	#########################################################

		TransmissionType for TxPDOs and RxPDOs:

			0:										Event controlled and sychron (with SYNC-Object)
			1-240:									Cyclic and synchron (with SYNC-Object)
			254:									Producer specified
			255:									Acyclic and eventcontrolled 
			255 and EventTime = InhibitTime:	Cyclic

	#########################################################	*)


	(*************************************************** TxPDOs of CANOpenSlave ( MOVI-PLC ReceiveObjects) ***********************************************************)

	ExtConfig.NumberOfTxPDO				:= 4;		(*  TxPDO ---> CANopenSlave Transmit *)

	ExtConfig.TxPDO[1].EventTime			:= 100;		(* Slave: Index 0x18xx SubIndex 5: CycleTime in ms for CANopenSlave TXPDO *)
	ExtConfig.TxPDO[1].InhibitTime			:= 10;		(* Slave: Index 0x18xx SubIndex 3: InhibitTime in ms for CANopenSlave TxPDO *)
	ExtConfig.TxPDO[1].TransmissionType	:= 255;		(* Slave: Index 0x18xx SubIndex 2: TransmissionType for this TxPDO *)

	ExtConfig.TxPDO[2].EventTime			:= 100;		(* Slave: Index 0x18xx SubIndex 5: CycleTime in ms for CANopenSlave TXPDO *)
	ExtConfig.TxPDO[2].InhibitTime			:= 10;		(* Slave: Index 0x18xx SubIndex 3: InhibitTime in ms for CANopenSlave TxPDO *)
	ExtConfig.TxPDO[2].TransmissionType	:= 255;		(* Slave: Index 0x18xx SubIndex 2: TransmissionType for this TxPDO *)

	ExtConfig.TxPDO[3].EventTime			:= 100;		(* Slave: Index 0x18xx SubIndex 5: CycleTime in ms for CANopenSlave TXPDO *)
	ExtConfig.TxPDO[3].InhibitTime			:= 10;		(* Slave: Index 0x18xx SubIndex 3: InhibitTime in ms for CANopenSlave TxPDO *)
	ExtConfig.TxPDO[3].TransmissionType	:= 255;		(* Slave: Index 0x18xx SubIndex 2: TransmissionType for this TxPDO *)

	ExtConfig.TxPDO[4].EventTime			:= 100;		(* Slave: Index 0x18xx SubIndex 5: CycleTime in ms for CANopenSlave TXPDO *)
	ExtConfig.TxPDO[4].InhibitTime			:= 10;		(* Slave: Index 0x18xx SubIndex 3: InhibitTime in ms for CANopenSlave TxPDO *)
	ExtConfig.TxPDO[4].TransmissionType	:= 255;		(* Slave: Index 0x18xx SubIndex 2: TransmissionType for this TxPDO *)


	(*************************************************** RxPDOs of CANOpenSlave ( MOVI-PLC TransmitObjects) **********************************************************)

	ExtConfig.NumberOfRxPDO				:= 4;		(*  RxPDO ---> CANopenSlave Receive *)

	ExtConfig.RxPDO[1].EventTime			:= 100;		(* Master: CycleTime in ms for TransmitObjects (MOVI-PLC) *)
	ExtConfig.RxPDO[1].InhibitTime			:= 10;		(* Master: InhibitTime in ms for TransmitObjects (MOVI-PLC) *)
	ExtConfig.RxPDO[1].Length				:= 8;		(* Master: Length of this TransmitObject in bytes *)
	ExtConfig.RxPDO[1].TransmissionType	:= 255;		(* Slave: Index 0x14xx SubIndex 2: TransmissionType for this RxPDO *)

	ExtConfig.RxPDO[2].EventTime			:= 100;		(* Master: CycleTime in ms for TransmitObjects (MOVI-PLC) *)
	ExtConfig.RxPDO[2].InhibitTime			:= 10;		(* Master: InhibitTime in ms for TransmitObjects (MOVI-PLC) *)
	ExtConfig.RxPDO[2].Length				:= 8;		(* Master: Length of this TransmitObject in bytes *)
	ExtConfig.RxPDO[2].TransmissionType	:= 255;		(* Slave: Index 0x14xx SubIndex 2: TransmissionType for this RxPDO *)

	ExtConfig.RxPDO[3].EventTime			:= 100;		(* Master: CycleTime in ms for TransmitObjects (MOVI-PLC) *)
	ExtConfig.RxPDO[3].InhibitTime			:= 10;		(* Master: InhibitTime in ms for TransmitObjects (MOVI-PLC) *)
	ExtConfig.RxPDO[3].Length				:= 8;		(* Master: Length of this TransmitObject in bytes *)
	ExtConfig.RxPDO[3].TransmissionType	:= 255;		(* Slave: Index 0x14xx SubIndex 2: TransmissionType for this RxPDO *)

	ExtConfig.RxPDO[4].EventTime			:= 100;		(* Master: CycleTime in ms for TransmitObjects (MOVI-PLC) *)
	ExtConfig.RxPDO[4].InhibitTime			:= 10;		(* Master: InhibitTime in ms for TransmitObjects (MOVI-PLC) *)
	ExtConfig.RxPDO[4].Length				:= 8;		(* Master: Length of this TransmitObject in bytes *)
	ExtConfig.RxPDO[4].TransmissionType	:= 255;		(* Slave: Index 0x14xx SubIndex 2: TransmissionType for this RxPDO *)


	(***************************************************** Additional parameters to set in the CANOpenSlave  ***************************************************************)
(* Parameter for Cube67 DIO16 (56601) Submodul *)
	ExtConfig.stInitialParameter_COSlave.aIndex[1]			:= 16#2002;(*2. Module*)
	ExtConfig.stInitialParameter_COSlave.aSubIndex[1]	:= 2;(* Input function *)
	ExtConfig.stInitialParameter_COSlave.aBytes[1]		:= 1;
	ExtConfig.stInitialParameter_COSlave.aData[1]			:= 2#00000000;(* 0=Input, 1=Diag Input *)

	ExtConfig.stInitialParameter_COSlave.aIndex[2]			:= 16#2002;(*2. Module*)
	ExtConfig.stInitialParameter_COSlave.aSubIndex[2]	:= 3;(* Inpu/Output selection, channel 0..7,  Pin4*)
	ExtConfig.stInitialParameter_COSlave.aBytes[2]		:= 1;
	ExtConfig.stInitialParameter_COSlave.aData[2]			:= 2#00000000;(* 0=Input, 1=Output *)

	ExtConfig.stInitialParameter_COSlave.aIndex[3]			:= 16#2002;(*2. Module*)
	ExtConfig.stInitialParameter_COSlave.aSubIndex[3]	:= 4;(* Inpu/Output selection, channel 10..17,  Pin2*)
	ExtConfig.stInitialParameter_COSlave.aBytes[3]		:= 1;
	ExtConfig.stInitialParameter_COSlave.aData[3]			:= 2#00000000;(* 0=Input, 1=Output *)

	ExtConfig.stInitialParameter_COSlave.aIndex[4]			:= 16#2002;(*2. Module*)
	ExtConfig.stInitialParameter_COSlave.aSubIndex[4]	:= 5;(*Failsafe Mode, channel 0..7,  Pin4*)
	ExtConfig.stInitialParameter_COSlave.aBytes[4]		:= 1;
	ExtConfig.stInitialParameter_COSlave.aData[4]			:= 2#00000000;(* 0=last state, 1=Failsafe value *)

	ExtConfig.stInitialParameter_COSlave.aIndex[5]			:= 16#2002;(*2. Module*)
	ExtConfig.stInitialParameter_COSlave.aSubIndex[5]	:= 6;(*Failsafe Mode, channel 10..17,  Pin2*)
	ExtConfig.stInitialParameter_COSlave.aBytes[5]		:= 1;
	ExtConfig.stInitialParameter_COSlave.aData[5]			:= 2#00000000;(* 0=last state, 1=Failsafe value *)

	ExtConfig.stInitialParameter_COSlave.aIndex[6]			:= 16#2002;(*2. Module*)
	ExtConfig.stInitialParameter_COSlave.aSubIndex[6]	:= 7;(*Failsafe Value, channel 0..7,  Pin4*)
	ExtConfig.stInitialParameter_COSlave.aBytes[6]		:= 1;
	ExtConfig.stInitialParameter_COSlave.aData[6]			:= 2#00000000;(* 0=output low, 1=output high *)

	ExtConfig.stInitialParameter_COSlave.aIndex[7]			:= 16#2002;(*2. Module*)
	ExtConfig.stInitialParameter_COSlave.aSubIndex[7]	:= 8;(*Failsafe Value, channel 10..17,  Pin2*)
	ExtConfig.stInitialParameter_COSlave.aBytes[7]		:= 1;
	ExtConfig.stInitialParameter_COSlave.aData[7]			:= 2#00000000;(* 0=output low, 1=output high *)

	ExtConfig.stInitialParameter_COSlave.aIndex[8]			:= 16#2002;(*2. Module*)
	ExtConfig.stInitialParameter_COSlave.aSubIndex[8]	:= 9;(*function, channel 0..7,  Pin4*)
	ExtConfig.stInitialParameter_COSlave.aBytes[8]		:= 1;
	ExtConfig.stInitialParameter_COSlave.aData[8]			:= 2#00000000;(* 0=input no, 1=input nc *)

	ExtConfig.stInitialParameter_COSlave.aIndex[9]			:= 16#2002;(*2. Module*)
	ExtConfig.stInitialParameter_COSlave.aSubIndex[9]	:= 10;(*function, channel 10..17,  Pin2*)
	ExtConfig.stInitialParameter_COSlave.aBytes[9]		:= 1;
	ExtConfig.stInitialParameter_COSlave.aData[9]			:= 2#00000000;(* 0=input no, 1=input nc *)

(* Parameter for Cube67 DIO8 (56610) Submodul *)
	ExtConfig.stInitialParameter_COSlave.aIndex[10]		:= 16#2003;(*3 Module*)
	ExtConfig.stInitialParameter_COSlave.aSubIndex[10]	:= 2;(* Input function *)
	ExtConfig.stInitialParameter_COSlave.aBytes[10]		:= 1;
	ExtConfig.stInitialParameter_COSlave.aData[10]		:= 2#0000;(* 0=Input, 1=Diag Input *)

	ExtConfig.stInitialParameter_COSlave.aIndex[11]		:= 16#2003;(*3 Module*)
	ExtConfig.stInitialParameter_COSlave.aSubIndex[11]	:= 3;(* Inpu/Output selection, channel 0..3  Pin4*)
	ExtConfig.stInitialParameter_COSlave.aBytes[11]		:= 1;
	ExtConfig.stInitialParameter_COSlave.aData[11]		:= 2#0000;(* 0=Input, 1=Output *)

	ExtConfig.stInitialParameter_COSlave.aIndex[12]		:= 16#2003;(*3. Module*)
	ExtConfig.stInitialParameter_COSlave.aSubIndex[12]	:= 4;(* Inpu/Output selection, channel 10..13  Pin2*)
	ExtConfig.stInitialParameter_COSlave.aBytes[12]		:= 1;
	ExtConfig.stInitialParameter_COSlave.aData[12]		:= 2#0000;(* 0=Input, 1=Output *)

	ExtConfig.stInitialParameter_COSlave.aIndex[13]		:= 16#2003;(*3. Module*)
	ExtConfig.stInitialParameter_COSlave.aSubIndex[13]	:= 5;(*Failsafe Mode, channel 0..3,  Pin4*)
	ExtConfig.stInitialParameter_COSlave.aBytes[13]		:= 1;
	ExtConfig.stInitialParameter_COSlave.aData[13]		:= 2#0000;(* 0=last state, 1=Failsafe value *)

	ExtConfig.stInitialParameter_COSlave.aIndex[14]		:= 16#2003;(*3. Module*)
	ExtConfig.stInitialParameter_COSlave.aSubIndex[14]	:= 6;(*Failsafe Mode, channel 10..13,  Pin2*)
	ExtConfig.stInitialParameter_COSlave.aBytes[14]		:= 1;
	ExtConfig.stInitialParameter_COSlave.aData[14]		:= 2#0000;(* 0=last state, 1=Failsafe value *)

	ExtConfig.stInitialParameter_COSlave.aIndex[15]		:= 16#2003;(*3. Module*)
	ExtConfig.stInitialParameter_COSlave.aSubIndex[15]	:= 7;(*Failsafe Value, channel 0..3,  Pin4*)
	ExtConfig.stInitialParameter_COSlave.aBytes[15]		:= 1;
	ExtConfig.stInitialParameter_COSlave.aData[15]		:= 2#0000;(* 0=output low, 1=output high *)

	ExtConfig.stInitialParameter_COSlave.aIndex[16]		:= 16#2003;(*3. Module*)
	ExtConfig.stInitialParameter_COSlave.aSubIndex[16]	:= 8;(*Failsafe Value, channel 10..13,  Pin2*)
	ExtConfig.stInitialParameter_COSlave.aBytes[16]		:= 1;
	ExtConfig.stInitialParameter_COSlave.aData[16]		:= 2#0000;(* 0=output low, 1=output high *)

	ExtConfig.stInitialParameter_COSlave.aIndex[17]		:= 16#2003;(*3. Module*)
	ExtConfig.stInitialParameter_COSlave.aSubIndex[17]	:= 9;(*function, channel 0..3,  Pin4*)
	ExtConfig.stInitialParameter_COSlave.aBytes[17]		:= 1;
	ExtConfig.stInitialParameter_COSlave.aData[17]		:= 2#0000;(* 0=input no, 1=input nc *)

	ExtConfig.stInitialParameter_COSlave.aIndex[18]		:= 16#2003;(*3. Module*)
	ExtConfig.stInitialParameter_COSlave.aSubIndex[18]	:= 10;(*function, channel 10..13,  Pin2*)
	ExtConfig.stInitialParameter_COSlave.aBytes[18]		:= 1;
	ExtConfig.stInitialParameter_COSlave.aData[18]		:= 2#0000;(* 0=input no, 1=input nc *)

(* Parameter for Cube67 DIO8/DI8 (56691) Submodul *)
	ExtConfig.stInitialParameter_COSlave.aIndex[19]		:= 16#2001;(*1. Module*)
	ExtConfig.stInitialParameter_COSlave.aSubIndex[19]	:= 1;(* Inpu/Output selection, channel 0..7*)
	ExtConfig.stInitialParameter_COSlave.aBytes[19]		:= 1;
	ExtConfig.stInitialParameter_COSlave.aData[19]		:= 2#00000010;(* 0=Input, 1=Output *)

	ExtConfig.stInitialParameter_COSlave.aIndex[20]		:= 16#2001;(*1.. Module*)
	ExtConfig.stInitialParameter_COSlave.aSubIndex[20]	:= 2;(*Failsafe Mode, channel 0..7*)
	ExtConfig.stInitialParameter_COSlave.aBytes[20]		:= 1;
	ExtConfig.stInitialParameter_COSlave.aData[20]		:= 2#0000;(* 0=last state, 1=Failsafe value *)

	ExtConfig.stInitialParameter_COSlave.aIndex[21]		:= 16#2001;(*1. Module*)
	ExtConfig.stInitialParameter_COSlave.aSubIndex[21]	:= 3;(*Failsafe Value, channel 0..7*)
	ExtConfig.stInitialParameter_COSlave.aBytes[21]		:= 1;
	ExtConfig.stInitialParameter_COSlave.aData[21]		:= 2#0000;(* 0=output low, 1=output high *)

	ExtConfig.stInitialParameter_COSlave.aIndex[22]		:= 16#2001;(*1. Module*)
	ExtConfig.stInitialParameter_COSlave.aSubIndex[22]	:= 4;(*function, channel 0..7*)
	ExtConfig.stInitialParameter_COSlave.aBytes[22]		:= 1;
	ExtConfig.stInitialParameter_COSlave.aData[22]		:= 2#0000;(* 0=input no, 1=input nc *)

	ExtConfig.stInitialParameter_COSlave.aIndex[23]		:= 16#2001;(*1. Module*)
	ExtConfig.stInitialParameter_COSlave.aSubIndex[23]	:= 5;(*function, channel 10..17*)
	ExtConfig.stInitialParameter_COSlave.aBytes[23]		:= 1;
	ExtConfig.stInitialParameter_COSlave.aData[23]		:= 2#0000;(* 0=input no, 1=input nc *)


(*	(* Enable transmission of analog inputs *)
	ExtConfig.stInitialParameter_COSlave.aIndex[24]		:= 16#6423;
	ExtConfig.stInitialParameter_COSlave.aSubIndex[24]	:= 0;
	ExtConfig.stInitialParameter_COSlave.aBytes[24]		:= 1;
	ExtConfig.stInitialParameter_COSlave.aData[24]		:= 1;
*)

(* Enable automatic PDO mapping *)
	ExtConfig.stInitialParameter_COSlave.aIndex[24]		:= 16#2100;
	ExtConfig.stInitialParameter_COSlave.aSubIndex[24]	:= 0;
	ExtConfig.stInitialParameter_COSlave.aBytes[24]		:= 1;
	ExtConfig.stInitialParameter_COSlave.aData[24]		:= 1;

	(********************************************** Additional configuration. Default values are in most cases sufficient *****************************************************)

	ExtConfig.bIOHold						:= FALSE;
	ExtConfig.bNoSettingsDownload			:= FALSE;
	ExtConfig.bWaitBeforeOperational		:= FALSE;
	ExtConfig.bResetUnconditional			:= FALSE;

	ExtConfig.TimeOutHeartBeat				:= 250;				(* [ms] *)
(*	ExtConfig.DivTimeOutHeartBeat			:= 2;				(* Heartbeat Consumer = ExtConfig.TimeOutHeartBeat	 / ExtConfig.DivTimeOutHeartBeat *)*)
	ExtConfig.TimeOutNodeGuarding		:= 0;				(* [ms]. CAUTION ! DHP11B (MOVI-PLC basic) does NOT support NodeGuarding *)
	ExtConfig.TimeOutInitSequence			:= 10;				(* [seconds]. If the Init-Sequence takes longer than this TimeOut time --> Error *)
	ExtConfig.SyncCOBID						:= 0;				(* SyncObject ID for TransmissionType 0-240 (RxPDO). Usually 128. If 0, the ID will not be written *)
	ExtConfig.SyncTime						:= 0;				(* CycleTime for the SYNC-Object *)

	ExtConfig.TxPDO[1].COBID				:= 16#180;			(* In order to disable the use of RTR frames for the PDOs, set bit 30 = "RTR not allowed" *)
	ExtConfig.TxPDO[2].COBID				:= 16#280;			(* Ex. 16#4000_0280 *)
	ExtConfig.TxPDO[3].COBID				:= 16#380;
	ExtConfig.TxPDO[4].COBID				:= 16#480;			(* NOTE! These values are base values. The input "Address" will automatically be added *)
	ExtConfig.TxPDO[5].COBID				:= 16#680;
	ExtConfig.TxPDO[6].COBID				:= 16#1C0;
	ExtConfig.TxPDO[7].COBID				:= 16#2C0;
	ExtConfig.TxPDO[8].COBID				:= 16#3C0;
	ExtConfig.TxPDO[9].COBID				:= 16#4C0;
	ExtConfig.TxPDO[10].COBID				:= 16#6C0;

	ExtConfig.RxPDO[1].COBID				:= 16#200;
	ExtConfig.RxPDO[2].COBID				:= 16#300;
	ExtConfig.RxPDO[3].COBID				:= 16#400;
	ExtConfig.RxPDO[4].COBID				:= 16#500;
	ExtConfig.RxPDO[5].COBID				:= 16#780;
	ExtConfig.RxPDO[6].COBID				:= 16#240;
	ExtConfig.RxPDO[7].COBID				:= 16#340;
	ExtConfig.RxPDO[8].COBID				:= 16#440;
	ExtConfig.RxPDO[9].COBID				:= 16#540;
	ExtConfig.RxPDO[10].COBID				:= 16#7C0;

	Done := TRUE;

END_IF
END_FUNCTION_BLOCK

(* POU CodeSamples/CANopen/UniversalMaster/FB_Configuration_CANopenSlave_Phoenix_FLS_CO_DI8, ST *)
FUNCTION_BLOCK FB_Configuration_CANopenSlave_Phoenix_FLS_CO_DI8
VAR_INPUT
	Enable: BOOL; 			(* Activate config *)
END_VAR
VAR_OUTPUT
	Done: BOOL;				(* Config done *)
END_VAR
VAR_IN_OUT
	ExtConfig : MC_EXTENDEDCONFIG_COSLAVE	;
	(*
		########################################################################################################
			MC_EXTENDEDCONFIG_COSLAVE
		#########################################################################################################

						
		Variable								Value			Description
		-------------------------------------------------------------------------------------------------------------------------------------------------------------
		bWaitBeforeOperational 				BOOL;			When TRUE, after the coupler has been parameterized, it won't be switched in operational
																before this variable is FALSE. This can be used for example, to store the configuration with the FB
																MPLC_Universal_CANopen, with Service "SEWIOS_STORE", after a reset of the coppler 
		-------------------------------------------------------------------------------------------------------------------------------------------------------------
		bNoSettingsDownload 				BOOL;			TRUE : No configuration of the module. The configuration has to be done manually.
		-------------------------------------------------------------------------------------------------------------------------------------------------------------
		bResetUnconditional 					BOOL;			Even if the Connect FB isn't in fault it is possible to reset the bus coppler
		-------------------------------------------------------------------------------------------------------------------------------------------------------------
		bIOHold 								BOOL;			TRUE : Input data remain unchanged and the output data are not resetet also if the FB is in fault 
		-------------------------------------------------------------------------------------------------------------------------------------------------------------
		TimeOutHeartBeat					UINT;			If this value (ms) is different to zero, HeartbeatMode will be activated
		-------------------------------------------------------------------------------------------------------------------------------------------------------------
		TimeOutNodeGuarding 				UINT;			If this value (ms) is different to zero, NodeGuarding will be activated. 
																Caution ! The MOVI-PLC basic doesn´t support NodeGuarding 
		-------------------------------------------------------------------------------------------------------------------------------------------------------------
		TimeOutInitSequence					UINT;			Timeout for initialisation sequence (seconds) 
		-------------------------------------------------------------------------------------------------------------------------------------------------------------
		NumberOfRxPDO 					UINT;			Receive PDO : MOVI-PLC --> Slave  max. 32 
		-------------------------------------------------------------------------------------------------------------------------------------------------------------
		NumberOfTxPDO 						UINT;			Send PDO :      Slave --> MOVI-PLC  max 32 
		-------------------------------------------------------------------------------------------------------------------------------------------------------------	
		SyncTime 								USINT;			Cycle time of the sync telegram in ms. 
																Default = 0 : no sync will be started.
																If  SyncTime > 0, this FB initializes a sync telegram with the ID set at SyncCOBID. 
																The slave has to support synchronous communication 
		-------------------------------------------------------------------------------------------------------------------------------------------------------------
		SyncCOBID							UINT;			Index 1005h. ID of the sync telegram. Usually 16#80. IF 0, the ID won't be written.
		-------------------------------------------------------------------------------------------------------------------------------------------------------------
		SyncTimeOut 							INT := -1;		Index 1006h. Normally equal to SyncTime. 
																The slave usually set SyncTimeOut equal to SyncTime * 1.5. 
																If < 0, the index won't be written. 0 means no control over the sync interval 
		-------------------------------------------------------------------------------------------------------------------------------------------------------------
		stInitialParameter_COSlave 			MC_INITIALPARAMETER_COSLAVE;
												(*#################################################################
												With this struct, user defined parameters will be written to the BusCoupler after the
												initialization of the MPLC_ConnectUniversalSlave_CANopen. 
												Add the following code to your program to initialise the struct : 
												Example:
												Index 16#6423:	Activates the event-driven transmission of PDOs with analog inputs
												Index 16#3500:	Index from the manufacturer specific profile area
	
													stInitialParameter_COSlave.aIndex[1] := 16#6423;  	(* Index to write to *)
													stInitialParameter_COSlave.aSubIndex[1] := 0;   	(* SubIndex to write to *)
													stInitialParameter_COSlave.aBytes[1] := 1;   		(* Number of bytes to write  *)
													stInitialParameter_COSlave.aData[1] := 1;   			(* Data *)
	
													stInitialParameter_COSlave.aIndex[2] := 16#3500;  	(* Index to write to *)
													stInitialParameter_COSlave.aSubIndex[2] := 0;   	(* SubIndex to write to *)
													stInitialParameter_COSlave.aBytes[2] := 2;   		(* Number of bytes to write *)
													stInitialParameter_COSlave.aData[2] := 5;   			(* Data *)
	
												If there are more than 10 (DHP11B) or 64 (DHx41B) parameters to write, declare 
												NUMOF_INITIALPARAMETER in your program.
	
													VAR_GLOBAL CONSTANT
														NUMOF_INITIALPARAMETER : UDINT := 20;	
													END_VAR
	
												##################################################################*)
			-------------------------------------------------------------------------------------------------------------------------------------------------------------
		(* IDs of the PDO telegrams. The IDs are always calculated with the following IDs as a basis + the address of the bus coupler *)

		RxPDO 								ARRAY[1..32] OF MC_PDO_COSLAVE;			(* MOVI-PLC --> Slave *)
												(* := 16#200,16#300,16#400,16#500,16#780,16#240,16#340,16#440,16#540,16#7C0;	*)
		-------------------------------------------------------------------------------------------------------------------------------------------------------------
		TxPDO 								ARRAY[1..32] OF MC_PDO_COSLAVE; 			(* Slave --> MOVI-PLC *)
												(*:= 16#180,16#280,16#380,16#480,16#680,16#1C0,16#2C0,16#3C0,16#4C0,16#6C0;*)
	*)
END_VAR
IF Enable AND NOT Done THEN

	(*########################################################

		Configuration of CANopenSlave (Phoenix FLS CO DI8)
		
	#########################################################

		TransmissionType for TxPDOs and RxPDOs:

			0:										Event controlled and sychron (with SYNC-Object)
			1-240:									Cyclic and synchron (with SYNC-Object)
			254:									Producer specified
			255:									Acyclic and eventcontrolled 
			255 and EventTime = InhibitTime:	Cyclic

	#########################################################	*)


	(*************************************************** TxPDOs of CANOpenSlave ( MOVI-PLC ReceiveObjects) ***********************************************************)

	ExtConfig.NumberOfTxPDO				:= 1;		(*  TxPDO ---> CANopenSlave Transmit *)

	ExtConfig.TxPDO[1].EventTime			:= 0;		(* Slave: Index 0x18xx SubIndex 5: CycleTime in ms for CANopenSlave TXPDO *)
	ExtConfig.TxPDO[1].InhibitTime			:= 0;		(* Slave: Index 0x18xx SubIndex 3: InhibitTime in ms for CANopenSlave TxPDO *)
	ExtConfig.TxPDO[1].TransmissionType	:= 255;		(* Slave: Index 0x18xx SubIndex 2: TransmissionType for this TxPDO *)


	(*************************************************** RxPDOs of CANOpenSlave ( MOVI-PLC TransmitObjects) **********************************************************)

	ExtConfig.NumberOfRxPDO				:= 0;		(*  RxPDO ---> CANopenSlave Receive *)

(*	ExtConfig.RxPDO[1].EventTime			:= 0;		(* Master: CycleTime in ms for TransmitObjects (MOVI-PLC) *)
	ExtConfig.RxPDO[1].InhibitTime			:= 0;		(* Master: InhibitTime in ms for TransmitObjects (MOVI-PLC) *)
	ExtConfig.RxPDO[1].Length				:= 1;		(* Master: Length of this TransmitObject in bytes *)
	ExtConfig.RxPDO[1].TransmissionType	:= 255;		(* Slave: Index 0x14xx SubIndex 2: TransmissionType for this RxPDO *)
*)

	(***************************************************** Additional parameters to set in the CANOpenSlave  ***************************************************************)

(*	Example to write user defined parameters (i.e. Index 16#6200):
	
	ExtConfig.stInitialParameter_COSlave.aIndex[1]			:= 16#6200;
	ExtConfig.stInitialParameter_COSlave.aSubIndex[1]	:= 0;
	ExtConfig.stInitialParameter_COSlave.aBytes[1]		:= 1;
	ExtConfig.stInitialParameter_COSlave.aData[1]			:= 16#64;
*)

	(********************************************** Additional configuration. Default values are in most cases sufficient *****************************************************)

	ExtConfig.bIOHold						:= FALSE;
	ExtConfig.bNoSettingsDownload			:= FALSE;
	ExtConfig.bWaitBeforeOperational		:= FALSE;
	ExtConfig.bResetUnconditional			:= FALSE;

	ExtConfig.TimeOutHeartBeat				:= 0;				(* [ms] *)
	ExtConfig.TimeOutNodeGuarding		:= 400;				(* [ms]. CAUTION ! DHP11B (MOVI-PLC basic) does NOT support NodeGuarding *)
	ExtConfig.TimeOutInitSequence			:= 6;				(* [seconds]. If the Init-Sequence takes longer than this TimeOut time --> Error *)
	ExtConfig.SyncCOBID						:= 0;				(* SyncObject ID for TransmissionType 0-240 (RxPDO). Usually 128. If 0, the ID will not be written *)
	ExtConfig.SyncTime						:= 0;				(* CycleTime for the SYNC-Object *)

	ExtConfig.TxPDO[1].COBID				:= 16#180;			(* In order to disable the use of RTR frames for the PDOs, set bit 30 = "RTR not allowed" *)
	ExtConfig.TxPDO[2].COBID				:= 16#280;			(* Ex. 16#4000_0280 *)
	ExtConfig.TxPDO[3].COBID				:= 16#380;
	ExtConfig.TxPDO[4].COBID				:= 16#480;			(* NOTE! These values are base values. The input "Address" will automatically be added *)
	ExtConfig.TxPDO[5].COBID				:= 16#680;
	ExtConfig.TxPDO[6].COBID				:= 16#1C0;
	ExtConfig.TxPDO[7].COBID				:= 16#2C0;
	ExtConfig.TxPDO[8].COBID				:= 16#3C0;
	ExtConfig.TxPDO[9].COBID				:= 16#4C0;
	ExtConfig.TxPDO[10].COBID				:= 16#6C0;

	ExtConfig.RxPDO[1].COBID				:= 16#200;
	ExtConfig.RxPDO[2].COBID				:= 16#300;
	ExtConfig.RxPDO[3].COBID				:= 16#400;
	ExtConfig.RxPDO[4].COBID				:= 16#500;
	ExtConfig.RxPDO[5].COBID				:= 16#780;
	ExtConfig.RxPDO[6].COBID				:= 16#240;
	ExtConfig.RxPDO[7].COBID				:= 16#340;
	ExtConfig.RxPDO[8].COBID				:= 16#440;
	ExtConfig.RxPDO[9].COBID				:= 16#540;
	ExtConfig.RxPDO[10].COBID				:= 16#7C0;

	Done := TRUE;

END_IF
END_FUNCTION_BLOCK

(* POU CodeSamples/CANopen/UniversalMaster/FB_Configuration_CANopenSlave_Phoenix_FLS_CO_DIO8_8, ST *)
FUNCTION_BLOCK FB_Configuration_CANopenSlave_Phoenix_FLS_CO_DIO8_8
VAR_INPUT
	Enable: BOOL; 			(* Activate config *)
END_VAR
VAR_OUTPUT
	Done: BOOL;				(* Config done *)
END_VAR
VAR_IN_OUT
	ExtConfig : MC_EXTENDEDCONFIG_COSLAVE	;
	(*
		########################################################################################################
			MC_EXTENDEDCONFIG_COSLAVE
		#########################################################################################################

						
		Variable								Value			Description
		-------------------------------------------------------------------------------------------------------------------------------------------------------------
		bWaitBeforeOperational 				BOOL;			When TRUE, after the coupler has been parameterized, it won't be switched in operational
																before this variable is FALSE. This can be used for example, to store the configuration with the FB
																MPLC_Universal_CANopen, with Service "SEWIOS_STORE", after a reset of the coppler 
		-------------------------------------------------------------------------------------------------------------------------------------------------------------
		bNoSettingsDownload 				BOOL;			TRUE : No configuration of the module. The configuration has to be done manually.
		-------------------------------------------------------------------------------------------------------------------------------------------------------------
		bResetUnconditional 					BOOL;			Even if the Connect FB isn't in fault it is possible to reset the bus coppler
		-------------------------------------------------------------------------------------------------------------------------------------------------------------
		bIOHold 								BOOL;			TRUE : Input data remain unchanged and the output data are not resetet also if the FB is in fault 
		-------------------------------------------------------------------------------------------------------------------------------------------------------------
		TimeOutHeartBeat					UINT;			If this value (ms) is different to zero, HeartbeatMode will be activated
		-------------------------------------------------------------------------------------------------------------------------------------------------------------
		TimeOutNodeGuarding 				UINT;			If this value (ms) is different to zero, NodeGuarding will be activated. 
																Caution ! The MOVI-PLC basic doesn´t support NodeGuarding 
		-------------------------------------------------------------------------------------------------------------------------------------------------------------
		TimeOutInitSequence					UINT;			Timeout for initialisation sequence (seconds) 
		-------------------------------------------------------------------------------------------------------------------------------------------------------------
		NumberOfRxPDO 					UINT;			Receive PDO : MOVI-PLC --> Slave  max. 32 
		-------------------------------------------------------------------------------------------------------------------------------------------------------------
		NumberOfTxPDO 						UINT;			Send PDO :      Slave --> MOVI-PLC  max 32 
		-------------------------------------------------------------------------------------------------------------------------------------------------------------	
		SyncTime 								USINT;			Cycle time of the sync telegram in ms. 
																Default = 0 : no sync will be started.
																If  SyncTime > 0, this FB initializes a sync telegram with the ID set at SyncCOBID. 
																The slave has to support synchronous communication 
		-------------------------------------------------------------------------------------------------------------------------------------------------------------
		SyncCOBID							UINT;			Index 1005h. ID of the sync telegram. Usually 16#80. IF 0, the ID won't be written.
		-------------------------------------------------------------------------------------------------------------------------------------------------------------
		SyncTimeOut 							INT := -1;		Index 1006h. Normally equal to SyncTime. 
																The slave usually set SyncTimeOut equal to SyncTime * 1.5. 
																If < 0, the index won't be written. 0 means no control over the sync interval 
		-------------------------------------------------------------------------------------------------------------------------------------------------------------
		stInitialParameter_COSlave 			MC_INITIALPARAMETER_COSLAVE;
												(*#################################################################
												With this struct, user defined parameters will be written to the BusCoupler after the
												initialization of the MPLC_ConnectUniversalSlave_CANopen. 
												Add the following code to your program to initialise the struct : 
												Example:
												Index 16#6423:	Activates the event-driven transmission of PDOs with analog inputs
												Index 16#3500:	Index from the manufacturer specific profile area
	
													stInitialParameter_COSlave.aIndex[1] := 16#6423;  	(* Index to write to *)
													stInitialParameter_COSlave.aSubIndex[1] := 0;   	(* SubIndex to write to *)
													stInitialParameter_COSlave.aBytes[1] := 1;   		(* Number of bytes to write  *)
													stInitialParameter_COSlave.aData[1] := 1;   			(* Data *)
	
													stInitialParameter_COSlave.aIndex[2] := 16#3500;  	(* Index to write to *)
													stInitialParameter_COSlave.aSubIndex[2] := 0;   	(* SubIndex to write to *)
													stInitialParameter_COSlave.aBytes[2] := 2;   		(* Number of bytes to write *)
													stInitialParameter_COSlave.aData[2] := 5;   			(* Data *)
	
												If there are more than 10 (DHP11B) or 64 (DHx41B) parameters to write, declare 
												NUMOF_INITIALPARAMETER in your program.
	
													VAR_GLOBAL CONSTANT
														NUMOF_INITIALPARAMETER : UDINT := 20;	
													END_VAR
	
												##################################################################*)
			-------------------------------------------------------------------------------------------------------------------------------------------------------------
		(* IDs of the PDO telegrams. The IDs are always calculated with the following IDs as a basis + the address of the bus coupler *)

		RxPDO 								ARRAY[1..32] OF MC_PDO_COSLAVE;			(* MOVI-PLC --> Slave *)
												(* := 16#200,16#300,16#400,16#500,16#780,16#240,16#340,16#440,16#540,16#7C0;	*)
		-------------------------------------------------------------------------------------------------------------------------------------------------------------
		TxPDO 								ARRAY[1..32] OF MC_PDO_COSLAVE; 			(* Slave --> MOVI-PLC *)
												(*:= 16#180,16#280,16#380,16#480,16#680,16#1C0,16#2C0,16#3C0,16#4C0,16#6C0;*)
	*)
END_VAR
IF Enable AND NOT Done THEN

	(*########################################################

		Configuration of CANopenSlave (Phoenix FLS CO DIO8/8)
		
	#########################################################

		TransmissionType for TxPDOs and RxPDOs:

			0:										Event controlled and sychron (with SYNC-Object)
			1-240:									Cyclic and synchron (with SYNC-Object)
			254:									Producer specified
			255:									Acyclic and eventcontrolled 
			255 and EventTime = InhibitTime:	Cyclic

	#########################################################	*)


	(*************************************************** TxPDOs of CANOpenSlave ( MOVI-PLC ReceiveObjects) ***********************************************************)

	ExtConfig.NumberOfTxPDO				:= 1;		(*  TxPDO ---> CANopenSlave Transmit *)

	ExtConfig.TxPDO[1].EventTime			:= 0;		(* Slave: Index 0x18xx SubIndex 5: CycleTime in ms for CANopenSlave TXPDO *)
	ExtConfig.TxPDO[1].InhibitTime			:= 0;		(* Slave: Index 0x18xx SubIndex 3: InhibitTime in ms for CANopenSlave TxPDO *)
	ExtConfig.TxPDO[1].TransmissionType	:= 255;		(* Slave: Index 0x18xx SubIndex 2: TransmissionType for this TxPDO *)


	(*************************************************** RxPDOs of CANOpenSlave ( MOVI-PLC TransmitObjects) **********************************************************)

	ExtConfig.NumberOfRxPDO				:= 1;		(*  RxPDO ---> CANopenSlave Receive *)

	ExtConfig.RxPDO[1].EventTime			:= 0;		(* Master: CycleTime in ms for TransmitObjects (MOVI-PLC) *)
	ExtConfig.RxPDO[1].InhibitTime			:= 0;		(* Master: InhibitTime in ms for TransmitObjects (MOVI-PLC) *)
	ExtConfig.RxPDO[1].Length				:= 1;		(* Master: Length of this TransmitObject in bytes *)
	ExtConfig.RxPDO[1].TransmissionType	:= 255;		(* Slave: Index 0x14xx SubIndex 2: TransmissionType for this RxPDO *)


	(***************************************************** Additional parameters to set in the CANOpenSlave  ***************************************************************)

(*	Example to write user defined parameters (i.e. Index 16#6200):
	
	ExtConfig.stInitialParameter_COSlave.aIndex[1]			:= 16#6200;
	ExtConfig.stInitialParameter_COSlave.aSubIndex[1]	:= 0;
	ExtConfig.stInitialParameter_COSlave.aBytes[1]		:= 1;
	ExtConfig.stInitialParameter_COSlave.aData[1]			:= 16#64;
*)

	(********************************************** Additional configuration. Default values are in most cases sufficient *****************************************************)

	ExtConfig.bIOHold						:= FALSE;
	ExtConfig.bNoSettingsDownload			:= FALSE;
	ExtConfig.bWaitBeforeOperational		:= FALSE;
	ExtConfig.bResetUnconditional			:= FALSE;

	ExtConfig.TimeOutHeartBeat				:= 0;				(* [ms] *)
	ExtConfig.TimeOutNodeGuarding		:= 400;				(* [ms]. CAUTION ! DHP11B (MOVI-PLC basic) does NOT support NodeGuarding *)
	ExtConfig.TimeOutInitSequence			:= 6;				(* [seconds]. If the Init-Sequence takes longer than this TimeOut time --> Error *)
	ExtConfig.SyncCOBID						:= 0;				(* SyncObject ID for TransmissionType 0-240 (RxPDO). Usually 128. If 0, the ID will not be written *)
	ExtConfig.SyncTime						:= 0;				(* CycleTime for the SYNC-Object *)

	ExtConfig.TxPDO[1].COBID				:= 16#180;			(* In order to disable the use of RTR frames for the PDOs, set bit 30 = "RTR not allowed" *)
	ExtConfig.TxPDO[2].COBID				:= 16#280;			(* Ex. 16#4000_0280 *)
	ExtConfig.TxPDO[3].COBID				:= 16#380;
	ExtConfig.TxPDO[4].COBID				:= 16#480;			(* NOTE! These values are base values. The input "Address" will automatically be added *)
	ExtConfig.TxPDO[5].COBID				:= 16#680;
	ExtConfig.TxPDO[6].COBID				:= 16#1C0;
	ExtConfig.TxPDO[7].COBID				:= 16#2C0;
	ExtConfig.TxPDO[8].COBID				:= 16#3C0;
	ExtConfig.TxPDO[9].COBID				:= 16#4C0;
	ExtConfig.TxPDO[10].COBID				:= 16#6C0;

	ExtConfig.RxPDO[1].COBID				:= 16#200;
	ExtConfig.RxPDO[2].COBID				:= 16#300;
	ExtConfig.RxPDO[3].COBID				:= 16#400;
	ExtConfig.RxPDO[4].COBID				:= 16#500;
	ExtConfig.RxPDO[5].COBID				:= 16#780;
	ExtConfig.RxPDO[6].COBID				:= 16#240;
	ExtConfig.RxPDO[7].COBID				:= 16#340;
	ExtConfig.RxPDO[8].COBID				:= 16#440;
	ExtConfig.RxPDO[9].COBID				:= 16#540;
	ExtConfig.RxPDO[10].COBID				:= 16#7C0;

	Done := TRUE;

END_IF
END_FUNCTION_BLOCK

(* POU CodeSamples/CANopen/UniversalMaster/FB_Configuration_CANopenSlave_Phoenix_FLS_CO_DO8, ST *)
FUNCTION_BLOCK FB_Configuration_CANopenSlave_Phoenix_FLS_CO_DO8
VAR_INPUT
	Enable: BOOL; 			(* Activate config *)
END_VAR
VAR_OUTPUT
	Done: BOOL;				(* Config done *)
END_VAR
VAR_IN_OUT
	ExtConfig : MC_EXTENDEDCONFIG_COSLAVE	;
	(*
		########################################################################################################
			MC_EXTENDEDCONFIG_COSLAVE
		#########################################################################################################

						
		Variable								Value			Description
		-------------------------------------------------------------------------------------------------------------------------------------------------------------
		bWaitBeforeOperational 				BOOL;			When TRUE, after the coupler has been parameterized, it won't be switched in operational
																before this variable is FALSE. This can be used for example, to store the configuration with the FB
																MPLC_Universal_CANopen, with Service "SEWIOS_STORE", after a reset of the coppler 
		-------------------------------------------------------------------------------------------------------------------------------------------------------------
		bNoSettingsDownload 				BOOL;			TRUE : No configuration of the module. The configuration has to be done manually.
		-------------------------------------------------------------------------------------------------------------------------------------------------------------
		bResetUnconditional 					BOOL;			Even if the Connect FB isn't in fault it is possible to reset the bus coppler
		-------------------------------------------------------------------------------------------------------------------------------------------------------------
		bIOHold 								BOOL;			TRUE : Input data remain unchanged and the output data are not resetet also if the FB is in fault 
		-------------------------------------------------------------------------------------------------------------------------------------------------------------
		TimeOutHeartBeat					UINT;			If this value (ms) is different to zero, HeartbeatMode will be activated
		-------------------------------------------------------------------------------------------------------------------------------------------------------------
		TimeOutNodeGuarding 				UINT;			If this value (ms) is different to zero, NodeGuarding will be activated. 
																Caution ! The MOVI-PLC basic doesn´t support NodeGuarding 
		-------------------------------------------------------------------------------------------------------------------------------------------------------------
		TimeOutInitSequence					UINT;			Timeout for initialisation sequence (seconds) 
		-------------------------------------------------------------------------------------------------------------------------------------------------------------
		NumberOfRxPDO 					UINT;			Receive PDO : MOVI-PLC --> Slave  max. 32 
		-------------------------------------------------------------------------------------------------------------------------------------------------------------
		NumberOfTxPDO 						UINT;			Send PDO :      Slave --> MOVI-PLC  max 32 
		-------------------------------------------------------------------------------------------------------------------------------------------------------------	
		SyncTime 								USINT;			Cycle time of the sync telegram in ms. 
																Default = 0 : no sync will be started.
																If  SyncTime > 0, this FB initializes a sync telegram with the ID set at SyncCOBID. 
																The slave has to support synchronous communication 
		-------------------------------------------------------------------------------------------------------------------------------------------------------------
		SyncCOBID							UINT;			Index 1005h. ID of the sync telegram. Usually 16#80. IF 0, the ID won't be written.
		-------------------------------------------------------------------------------------------------------------------------------------------------------------
		SyncTimeOut 							INT := -1;		Index 1006h. Normally equal to SyncTime. 
																The slave usually set SyncTimeOut equal to SyncTime * 1.5. 
																If < 0, the index won't be written. 0 means no control over the sync interval 
		-------------------------------------------------------------------------------------------------------------------------------------------------------------
		stInitialParameter_COSlave 			MC_INITIALPARAMETER_COSLAVE;
												(*#################################################################
												With this struct, user defined parameters will be written to the BusCoupler after the
												initialization of the MPLC_ConnectUniversalSlave_CANopen. 
												Add the following code to your program to initialise the struct : 
												Example:
												Index 16#6423:	Activates the event-driven transmission of PDOs with analog inputs
												Index 16#3500:	Index from the manufacturer specific profile area
	
													stInitialParameter_COSlave.aIndex[1] := 16#6423;  	(* Index to write to *)
													stInitialParameter_COSlave.aSubIndex[1] := 0;   	(* SubIndex to write to *)
													stInitialParameter_COSlave.aBytes[1] := 1;   		(* Number of bytes to write  *)
													stInitialParameter_COSlave.aData[1] := 1;   			(* Data *)
	
													stInitialParameter_COSlave.aIndex[2] := 16#3500;  	(* Index to write to *)
													stInitialParameter_COSlave.aSubIndex[2] := 0;   	(* SubIndex to write to *)
													stInitialParameter_COSlave.aBytes[2] := 2;   		(* Number of bytes to write *)
													stInitialParameter_COSlave.aData[2] := 5;   			(* Data *)
	
												If there are more than 10 (DHP11B) or 64 (DHx41B) parameters to write, declare 
												NUMOF_INITIALPARAMETER in your program.
	
													VAR_GLOBAL CONSTANT
														NUMOF_INITIALPARAMETER : UDINT := 20;	
													END_VAR
	
												##################################################################*)
			-------------------------------------------------------------------------------------------------------------------------------------------------------------
		(* IDs of the PDO telegrams. The IDs are always calculated with the following IDs as a basis + the address of the bus coupler *)

		RxPDO 								ARRAY[1..32] OF MC_PDO_COSLAVE;			(* MOVI-PLC --> Slave *)
												(* := 16#200,16#300,16#400,16#500,16#780,16#240,16#340,16#440,16#540,16#7C0;	*)
		-------------------------------------------------------------------------------------------------------------------------------------------------------------
		TxPDO 								ARRAY[1..32] OF MC_PDO_COSLAVE; 			(* Slave --> MOVI-PLC *)
												(*:= 16#180,16#280,16#380,16#480,16#680,16#1C0,16#2C0,16#3C0,16#4C0,16#6C0;*)
	*)
END_VAR
IF Enable AND NOT Done THEN

	(*########################################################

		Configuration of CANopenSlave (Phoenix FLS CO DO8)
		
	#########################################################

		TransmissionType for TxPDOs and RxPDOs:

			0:										Event controlled and sychron (with SYNC-Object)
			1-240:									Cyclic and synchron (with SYNC-Object)
			254:									Producer specified
			255:									Acyclic and eventcontrolled 
			255 and EventTime = InhibitTime:	Cyclic

	#########################################################	*)


	(*************************************************** TxPDOs of CANOpenSlave ( MOVI-PLC ReceiveObjects) ***********************************************************)

	ExtConfig.NumberOfTxPDO				:= 0;		(*  TxPDO ---> CANopenSlave Transmit *)

(*	ExtConfig.TxPDO[1].EventTime			:= 0;		(* Slave: Index 0x18xx SubIndex 5: CycleTime in ms for CANopenSlave TXPDO *)
	ExtConfig.TxPDO[1].InhibitTime			:= 0;		(* Slave: Index 0x18xx SubIndex 3: InhibitTime in ms for CANopenSlave TxPDO *)
	ExtConfig.TxPDO[1].TransmissionType	:= 255;		(* Slave: Index 0x18xx SubIndex 2: TransmissionType for this TxPDO *)
*)

	(*************************************************** RxPDOs of CANOpenSlave ( MOVI-PLC TransmitObjects) **********************************************************)

	ExtConfig.NumberOfRxPDO				:= 1;		(*  RxPDO ---> CANopenSlave Receive *)

	ExtConfig.RxPDO[1].EventTime			:= 0;		(* Master: CycleTime in ms for TransmitObjects (MOVI-PLC) *)
	ExtConfig.RxPDO[1].InhibitTime			:= 0;		(* Master: InhibitTime in ms for TransmitObjects (MOVI-PLC) *)
	ExtConfig.RxPDO[1].Length				:= 1;		(* Master: Length of this TransmitObject in bytes *)
	ExtConfig.RxPDO[1].TransmissionType	:= 255;		(* Slave: Index 0x14xx SubIndex 2: TransmissionType for this RxPDO *)


	(***************************************************** Additional parameters to set in the CANOpenSlave  ***************************************************************)

(*	Example to write user defined parameters (i.e. Index 16#6200):
	
	ExtConfig.stInitialParameter_COSlave.aIndex[1]			:= 16#6200;
	ExtConfig.stInitialParameter_COSlave.aSubIndex[1]	:= 0;
	ExtConfig.stInitialParameter_COSlave.aBytes[1]		:= 1;
	ExtConfig.stInitialParameter_COSlave.aData[1]			:= 16#64;
*)

	(********************************************** Additional configuration. Default values are in most cases sufficient *****************************************************)

	ExtConfig.bIOHold						:= FALSE;
	ExtConfig.bNoSettingsDownload			:= FALSE;
	ExtConfig.bWaitBeforeOperational		:= FALSE;
	ExtConfig.bResetUnconditional			:= FALSE;

	ExtConfig.TimeOutHeartBeat				:= 0;				(* [ms] *)
	ExtConfig.TimeOutNodeGuarding		:= 400;				(* [ms]. CAUTION ! DHP11B (MOVI-PLC basic) does NOT support NodeGuarding *)
	ExtConfig.TimeOutInitSequence			:= 6;				(* [seconds]. If the Init-Sequence takes longer than this TimeOut time --> Error *)
	ExtConfig.SyncCOBID						:= 0;				(* SyncObject ID for TransmissionType 0-240 (RxPDO). Usually 128. If 0, the ID will not be written *)
	ExtConfig.SyncTime						:= 0;				(* CycleTime for the SYNC-Object *)

	ExtConfig.TxPDO[1].COBID				:= 16#180;			(* In order to disable the use of RTR frames for the PDOs, set bit 30 = "RTR not allowed" *)
	ExtConfig.TxPDO[2].COBID				:= 16#280;			(* Ex. 16#4000_0280 *)
	ExtConfig.TxPDO[3].COBID				:= 16#380;
	ExtConfig.TxPDO[4].COBID				:= 16#480;			(* NOTE! These values are base values. The input "Address" will automatically be added *)
	ExtConfig.TxPDO[5].COBID				:= 16#680;
	ExtConfig.TxPDO[6].COBID				:= 16#1C0;
	ExtConfig.TxPDO[7].COBID				:= 16#2C0;
	ExtConfig.TxPDO[8].COBID				:= 16#3C0;
	ExtConfig.TxPDO[9].COBID				:= 16#4C0;
	ExtConfig.TxPDO[10].COBID				:= 16#6C0;

	ExtConfig.RxPDO[1].COBID				:= 16#200;
	ExtConfig.RxPDO[2].COBID				:= 16#300;
	ExtConfig.RxPDO[3].COBID				:= 16#400;
	ExtConfig.RxPDO[4].COBID				:= 16#500;
	ExtConfig.RxPDO[5].COBID				:= 16#780;
	ExtConfig.RxPDO[6].COBID				:= 16#240;
	ExtConfig.RxPDO[7].COBID				:= 16#340;
	ExtConfig.RxPDO[8].COBID				:= 16#440;
	ExtConfig.RxPDO[9].COBID				:= 16#540;
	ExtConfig.RxPDO[10].COBID				:= 16#7C0;

	Done := TRUE;

END_IF
END_FUNCTION_BLOCK

(* POU CodeSamples/CANopen/UniversalMaster/FB_Configuration_CANopenSlave_Phoenix_IL_CAN_BK_TC, ST *)
FUNCTION_BLOCK FB_Configuration_CANopenSlave_Phoenix_IL_CAN_BK_TC
VAR_INPUT
	Enable: BOOL; 			(* Activate config *)
END_VAR
VAR_OUTPUT
	Done: BOOL;				(* Config done *)
END_VAR
VAR_IN_OUT
	ExtConfig : MC_EXTENDEDCONFIG_COSLAVE	;
	(*
		########################################################################################################
			MC_EXTENDEDCONFIG_COSLAVE
		#########################################################################################################

						
		Variable								Value			Description
		-------------------------------------------------------------------------------------------------------------------------------------------------------------
		bWaitBeforeOperational 				BOOL;			When TRUE, after the coupler has been parameterized, it won't be switched in operational
																before this variable is FALSE. This can be used for example, to store the configuration with the FB
																MPLC_Universal_CANopen, with Service "SEWIOS_STORE", after a reset of the coppler 
		-------------------------------------------------------------------------------------------------------------------------------------------------------------
		bNoSettingsDownload 				BOOL;			TRUE : No configuration of the module. The configuration has to be done manually.
		-------------------------------------------------------------------------------------------------------------------------------------------------------------
		bResetUnconditional 					BOOL;			Even if the Connect FB isn't in fault it is possible to reset the bus coppler
		-------------------------------------------------------------------------------------------------------------------------------------------------------------
		bIOHold 								BOOL;			TRUE : Input data remain unchanged and the output data are not resetet also if the FB is in fault 
		-------------------------------------------------------------------------------------------------------------------------------------------------------------
		TimeOutHeartBeat					UINT;			If this value (ms) is different to zero, HeartbeatMode will be activated
		-------------------------------------------------------------------------------------------------------------------------------------------------------------
		TimeOutNodeGuarding 				UINT;			If this value (ms) is different to zero, NodeGuarding will be activated. 
																Caution ! The MOVI-PLC basic doesn´t support NodeGuarding 
		-------------------------------------------------------------------------------------------------------------------------------------------------------------
		TimeOutInitSequence					UINT;			Timeout for initialisation sequence (seconds) 
		-------------------------------------------------------------------------------------------------------------------------------------------------------------
		NumberOfRxPDO 					UINT;			Receive PDO : MOVI-PLC --> Slave  max. 32 
		-------------------------------------------------------------------------------------------------------------------------------------------------------------
		NumberOfTxPDO 						UINT;			Send PDO :      Slave --> MOVI-PLC  max 32 
		-------------------------------------------------------------------------------------------------------------------------------------------------------------	
		SyncTime 								USINT;			Cycle time of the sync telegram in ms. 
																Default = 0 : no sync will be started.
																If  SyncTime > 0, this FB initializes a sync telegram with the ID set at SyncCOBID. 
																The slave has to support synchronous communication 
		-------------------------------------------------------------------------------------------------------------------------------------------------------------
		SyncCOBID							UINT;			Index 1005h. ID of the sync telegram. Usually 16#80. IF 0, the ID won't be written.
		-------------------------------------------------------------------------------------------------------------------------------------------------------------
		SyncTimeOut 							INT := -1;		Index 1006h. Normally equal to SyncTime. 
																The slave usually set SyncTimeOut equal to SyncTime * 1.5. 
																If < 0, the index won't be written. 0 means no control over the sync interval 
		-------------------------------------------------------------------------------------------------------------------------------------------------------------
		stInitialParameter_COSlave 			MC_INITIALPARAMETER_COSLAVE;
												(*#################################################################
												With this struct, user defined parameters will be written to the BusCoupler after the
												initialization of the MPLC_ConnectUniversalSlave_CANopen. 
												Add the following code to your program to initialise the struct : 
												Example:
												Index 16#6423:	Activates the event-driven transmission of PDOs with analog inputs
												Index 16#3500:	Index from the manufacturer specific profile area
	
													stInitialParameter_COSlave.aIndex[1] := 16#6423;  	(* Index to write to *)
													stInitialParameter_COSlave.aSubIndex[1] := 0;   	(* SubIndex to write to *)
													stInitialParameter_COSlave.aBytes[1] := 1;   		(* Number of bytes to write  *)
													stInitialParameter_COSlave.aData[1] := 1;   			(* Data *)
	
													stInitialParameter_COSlave.aIndex[2] := 16#3500;  	(* Index to write to *)
													stInitialParameter_COSlave.aSubIndex[2] := 0;   	(* SubIndex to write to *)
													stInitialParameter_COSlave.aBytes[2] := 2;   		(* Number of bytes to write *)
													stInitialParameter_COSlave.aData[2] := 5;   			(* Data *)
	
												If there are more than 10 (DHP11B) or 64 (DHx41B) parameters to write, declare 
												NUMOF_INITIALPARAMETER in your program.
	
													VAR_GLOBAL CONSTANT
														NUMOF_INITIALPARAMETER : UDINT := 20;	
													END_VAR
	
												##################################################################*)
			-------------------------------------------------------------------------------------------------------------------------------------------------------------
		(* IDs of the PDO telegrams. The IDs are always calculated with the following IDs as a basis + the address of the bus coupler *)

		RxPDO 								ARRAY[1..32] OF MC_PDO_COSLAVE;			(* MOVI-PLC --> Slave *)
												(* := 16#200,16#300,16#400,16#500,16#780,16#240,16#340,16#440,16#540,16#7C0;	*)
		-------------------------------------------------------------------------------------------------------------------------------------------------------------
		TxPDO 								ARRAY[1..32] OF MC_PDO_COSLAVE; 			(* Slave --> MOVI-PLC *)
												(*:= 16#180,16#280,16#380,16#480,16#680,16#1C0,16#2C0,16#3C0,16#4C0,16#6C0;*)
	*)
END_VAR
IF Enable AND NOT Done THEN

	(*########################################################

		Configuration of CANopenSlave (Phoenix IL CAN BK TC)
		
	#########################################################

		TransmissionType for TxPDOs and RxPDOs:

			0:										Event controlled and sychron (with SYNC-Object)
			1-240:									Cyclic and synchron (with SYNC-Object)
			254:									Producer specified
			255:									Acyclic and eventcontrolled 
			255 and EventTime = InhibitTime:	Cyclic

	#########################################################	*)


	(*************************************************** TxPDOs of CANOpenSlave ( MOVI-PLC ReceiveObjects) ***********************************************************)

	ExtConfig.NumberOfTxPDO				:= 2;		(*  TxPDO ---> CANopenSlave Transmit *)

	ExtConfig.TxPDO[1].EventTime			:= 200;		(* Slave: Index 0x18xx SubIndex 5: CycleTime in ms for CANopenSlave TXPDO *)
	ExtConfig.TxPDO[1].InhibitTime			:= 5;		(* Slave: Index 0x18xx SubIndex 3: InhibitTime in ms for CANopenSlave TxPDO *)
	ExtConfig.TxPDO[1].TransmissionType	:= 255;		(* Slave: Index 0x18xx SubIndex 2: TransmissionType for this TxPDO *)

	ExtConfig.TxPDO[2].EventTime			:= 100;		(* Slave: Index 0x18xx SubIndex 5: CycleTime in ms for CANopenSlave TXPDO *)
	ExtConfig.TxPDO[2].InhibitTime			:= 100;		(* Slave: Index 0x18xx SubIndex 3: InhibitTime in ms for CANopenSlave TxPDO *)
	ExtConfig.TxPDO[2].TransmissionType	:= 255;		(* Slave: Index 0x18xx SubIndex 2: TransmissionType for this TxPDO *)


	(*************************************************** RxPDOs of CANOpenSlave ( MOVI-PLC TransmitObjects) **********************************************************)

	ExtConfig.NumberOfRxPDO				:= 2 (*3*);	(*  RxPDO ---> CANopenSlave Receive *)

	ExtConfig.RxPDO[1].EventTime			:= 200;		(* Master: CycleTime in ms for TransmitObjects (MOVI-PLC) *)
	ExtConfig.RxPDO[1].InhibitTime			:= 5;		(* Master: InhibitTime in ms for TransmitObjects (MOVI-PLC) *)
	ExtConfig.RxPDO[1].Length				:= 8;		(* Master: Length of this TransmitObject in bytes *)
	ExtConfig.RxPDO[1].TransmissionType	:= 255;		(* Slave: Index 0x14xx SubIndex 2: TransmissionType for this RxPDO *)

	ExtConfig.RxPDO[2].EventTime			:= 100;		(* Master: CycleTime in ms for TransmitObjects (MOVI-PLC) *)
	ExtConfig.RxPDO[2].InhibitTime			:= 100;		(* Master: InhibitTime in ms for TransmitObjects (MOVI-PLC) *)
	ExtConfig.RxPDO[2].Length				:= 8;		(* Master: Length of this TransmitObject in bytes *)
	ExtConfig.RxPDO[2].TransmissionType	:= 255;		(* Slave: Index 0x14xx SubIndex 2: TransmissionType for this RxPDO *)

(*	(* Special mapping for RxPDO3 *)
	ExtConfig.RxPDO[3].EventTime			:= 200;		(* Master: CycleTime in ms for TransmitObjects (MOVI-PLC) *)
	ExtConfig.RxPDO[3].InhibitTime			:= 5;		(* Master: InhibitTime in ms for TransmitObjects (MOVI-PLC) *)
	ExtConfig.RxPDO[3].Length				:= 2;		(* Master: Length of this TransmitObject in bytes *)
	ExtConfig.RxPDO[3].TransmissionType	:= 255;		(* Slave: Index 0x14xx SubIndex 2: TransmissionType for this RxPDO *)
*)

	(***************************************************** Additional parameters to set in the CANOpenSlave  ***************************************************************)

	(* Example of special mapping for RxPDO3 *)
	(* ################################ *)

(*	(* Deactivate PDO3 *)
	ExtConfig.stInitialParameter_COSlave.aIndex[1]			:= 16#1402;
	ExtConfig.stInitialParameter_COSlave.aSubIndex[1]	:= 1;
	ExtConfig.stInitialParameter_COSlave.aBytes[1]		:= 4;
	ExtConfig.stInitialParameter_COSlave.aData[1]			:= 16#8000_0000;

	(* Deactivate mapping for PDO3 *)
	ExtConfig.stInitialParameter_COSlave.aIndex[2]			:= 16#1602;
	ExtConfig.stInitialParameter_COSlave.aSubIndex[2]	:= 0;
	ExtConfig.stInitialParameter_COSlave.aBytes[2]		:= 1;
	ExtConfig.stInitialParameter_COSlave.aData[2]			:= 0;

	(* Map PDO3 Byte 1 *)
	ExtConfig.stInitialParameter_COSlave.aIndex[3]			:= 16#1602;
	ExtConfig.stInitialParameter_COSlave.aSubIndex[3]	:= 1;
	ExtConfig.stInitialParameter_COSlave.aBytes[3]		:= 4;
	ExtConfig.stInitialParameter_COSlave.aData[3]			:= 16#6200_09_08;

	(* Map PDO3 Byte 2 *)
	ExtConfig.stInitialParameter_COSlave.aIndex[4]			:= 16#1602;
	ExtConfig.stInitialParameter_COSlave.aSubIndex[4]	:= 2;
	ExtConfig.stInitialParameter_COSlave.aBytes[4]		:= 4;
	ExtConfig.stInitialParameter_COSlave.aData[4]			:= 16#6200_0A_08;

	(* Activate mapping for PDO3 *)
	ExtConfig.stInitialParameter_COSlave.aIndex[5]			:= 16#1602;
	ExtConfig.stInitialParameter_COSlave.aSubIndex[5]	:= 0;
	ExtConfig.stInitialParameter_COSlave.aBytes[5]		:= 1;
	ExtConfig.stInitialParameter_COSlave.aData[5]			:= 2;

	(* Activate PDO3 *)
	ExtConfig.stInitialParameter_COSlave.aIndex[6]			:= 16#1402;
	ExtConfig.stInitialParameter_COSlave.aSubIndex[6]	:= 1;
	ExtConfig.stInitialParameter_COSlave.aBytes[6]		:= 4;
	ExtConfig.stInitialParameter_COSlave.aData[6]			:= 16#0000_0403;
*)

	(********************************************** Additional configuration. Default values are in most cases sufficient *****************************************************)

	ExtConfig.bIOHold						:= FALSE;
	ExtConfig.bNoSettingsDownload			:= FALSE;
	ExtConfig.bWaitBeforeOperational		:= FALSE;
	ExtConfig.bResetUnconditional			:= FALSE;

	ExtConfig.TimeOutHeartBeat				:= 400;				(* [ms] *)
	ExtConfig.TimeOutNodeGuarding		:= 0;				(* [ms]. CAUTION ! DHP11B (MOVI-PLC basic) does NOT support NodeGuarding *)
	ExtConfig.TimeOutInitSequence			:= 10;				(* [seconds]. If the Init-Sequence takes longer than this TimeOut time --> Error *)
	ExtConfig.SyncCOBID						:= 0;				(* SyncObject ID for TransmissionType 0-240 (RxPDO). Usually 128. If 0, the ID will not be written *)
	ExtConfig.SyncTime						:= 0;				(* CycleTime for the SYNC-Object *)

	ExtConfig.TxPDO[1].COBID				:= 16#180;			(* In order to disable the use of RTR frames for the PDOs, set bit 30 = "RTR not allowed" *)
	ExtConfig.TxPDO[2].COBID				:= 16#280;			(* Ex. 16#4000_0280 *)
	ExtConfig.TxPDO[3].COBID				:= 16#380;
	ExtConfig.TxPDO[4].COBID				:= 16#480;			(* NOTE! These values are base values. The input "Address" will automatically be added *)
	ExtConfig.TxPDO[5].COBID				:= 16#680;
	ExtConfig.TxPDO[6].COBID				:= 16#1C0;
	ExtConfig.TxPDO[7].COBID				:= 16#2C0;
	ExtConfig.TxPDO[8].COBID				:= 16#3C0;
	ExtConfig.TxPDO[9].COBID				:= 16#4C0;
	ExtConfig.TxPDO[10].COBID				:= 16#6C0;

	ExtConfig.RxPDO[1].COBID				:= 16#200;
	ExtConfig.RxPDO[2].COBID				:= 16#300;
	ExtConfig.RxPDO[3].COBID				:= 16#400;
	ExtConfig.RxPDO[4].COBID				:= 16#500;
	ExtConfig.RxPDO[5].COBID				:= 16#780;
	ExtConfig.RxPDO[6].COBID				:= 16#240;
	ExtConfig.RxPDO[7].COBID				:= 16#340;
	ExtConfig.RxPDO[8].COBID				:= 16#440;
	ExtConfig.RxPDO[9].COBID				:= 16#540;
	ExtConfig.RxPDO[10].COBID				:= 16#7C0;

	Done := TRUE;

END_IF
END_FUNCTION_BLOCK

(* POU CodeSamples/CANopen/UniversalMaster/FB_Configuration_CANopenSlave_Phoenix_ILB_CO_DI16_DO16, ST *)
FUNCTION_BLOCK FB_Configuration_CANopenSlave_Phoenix_ILB_CO_DI16_DO16
VAR_INPUT
	Enable: BOOL; 			(* Activate config *)
END_VAR
VAR_OUTPUT
	Done: BOOL;				(* Config done *)
END_VAR
VAR_IN_OUT
	ExtConfig : MC_EXTENDEDCONFIG_COSLAVE	;
	(*
		########################################################################################################
			MC_EXTENDEDCONFIG_COSLAVE
		#########################################################################################################

						
		Variable								Value			Description
		-------------------------------------------------------------------------------------------------------------------------------------------------------------
		bWaitBeforeOperational 				BOOL;			When TRUE, after the coupler has been parameterized, it won't be switched in operational
																before this variable is FALSE. This can be used for example, to store the configuration with the FB
																MPLC_Universal_CANopen, with Service "SEWIOS_STORE", after a reset of the coppler 
		-------------------------------------------------------------------------------------------------------------------------------------------------------------
		bNoSettingsDownload 				BOOL;			TRUE : No configuration of the module. The configuration has to be done manually.
		-------------------------------------------------------------------------------------------------------------------------------------------------------------
		bResetUnconditional 					BOOL;			Even if the Connect FB isn't in fault it is possible to reset the bus coppler
		-------------------------------------------------------------------------------------------------------------------------------------------------------------
		bIOHold 								BOOL;			TRUE : Input data remain unchanged and the output data are not resetet also if the FB is in fault 
		-------------------------------------------------------------------------------------------------------------------------------------------------------------
		TimeOutHeartBeat					UINT;			If this value (ms) is different to zero, HeartbeatMode will be activated
		-------------------------------------------------------------------------------------------------------------------------------------------------------------
		TimeOutNodeGuarding 				UINT;			If this value (ms) is different to zero, NodeGuarding will be activated. 
																Caution ! The MOVI-PLC basic doesn´t support NodeGuarding 
		-------------------------------------------------------------------------------------------------------------------------------------------------------------
		TimeOutInitSequence					UINT;			Timeout for initialisation sequence (seconds) 
		-------------------------------------------------------------------------------------------------------------------------------------------------------------
		NumberOfRxPDO 					UINT;			Receive PDO : MOVI-PLC --> Slave  max. 32 
		-------------------------------------------------------------------------------------------------------------------------------------------------------------
		NumberOfTxPDO 						UINT;			Send PDO :      Slave --> MOVI-PLC  max 32 
		-------------------------------------------------------------------------------------------------------------------------------------------------------------	
		SyncTime 								USINT;			Cycle time of the sync telegram in ms. 
																Default = 0 : no sync will be started.
																If  SyncTime > 0, this FB initializes a sync telegram with the ID set at SyncCOBID. 
																The slave has to support synchronous communication 
		-------------------------------------------------------------------------------------------------------------------------------------------------------------
		SyncCOBID							UINT;			Index 1005h. ID of the sync telegram. Usually 16#80. IF 0, the ID won't be written.
		-------------------------------------------------------------------------------------------------------------------------------------------------------------
		SyncTimeOut 							INT := -1;		Index 1006h. Normally equal to SyncTime. 
																The slave usually set SyncTimeOut equal to SyncTime * 1.5. 
																If < 0, the index won't be written. 0 means no control over the sync interval 
		-------------------------------------------------------------------------------------------------------------------------------------------------------------
		stInitialParameter_COSlave 			MC_INITIALPARAMETER_COSLAVE;
												(*#################################################################
												With this struct, user defined parameters will be written to the BusCoupler after the
												initialization of the MPLC_ConnectUniversalSlave_CANopen. 
												Add the following code to your program to initialise the struct : 
												Example:
												Index 16#6423:	Activates the event-driven transmission of PDOs with analog inputs
												Index 16#3500:	Index from the manufacturer specific profile area
	
													stInitialParameter_COSlave.aIndex[1] := 16#6423;  	(* Index to write to *)
													stInitialParameter_COSlave.aSubIndex[1] := 0;   	(* SubIndex to write to *)
													stInitialParameter_COSlave.aBytes[1] := 1;   		(* Number of bytes to write  *)
													stInitialParameter_COSlave.aData[1] := 1;   			(* Data *)
	
													stInitialParameter_COSlave.aIndex[2] := 16#3500;  	(* Index to write to *)
													stInitialParameter_COSlave.aSubIndex[2] := 0;   	(* SubIndex to write to *)
													stInitialParameter_COSlave.aBytes[2] := 2;   		(* Number of bytes to write *)
													stInitialParameter_COSlave.aData[2] := 5;   			(* Data *)
	
												If there are more than 10 (DHP11B) or 64 (DHx41B) parameters to write, declare 
												NUMOF_INITIALPARAMETER in your program.
	
													VAR_GLOBAL CONSTANT
														NUMOF_INITIALPARAMETER : UDINT := 20;	
													END_VAR
	
												##################################################################*)
			-------------------------------------------------------------------------------------------------------------------------------------------------------------
		(* IDs of the PDO telegrams. The IDs are always calculated with the following IDs as a basis + the address of the bus coupler *)

		RxPDO 								ARRAY[1..32] OF MC_PDO_COSLAVE;			(* MOVI-PLC --> Slave *)
												(* := 16#200,16#300,16#400,16#500,16#780,16#240,16#340,16#440,16#540,16#7C0;	*)
		-------------------------------------------------------------------------------------------------------------------------------------------------------------
		TxPDO 								ARRAY[1..32] OF MC_PDO_COSLAVE; 			(* Slave --> MOVI-PLC *)
												(*:= 16#180,16#280,16#380,16#480,16#680,16#1C0,16#2C0,16#3C0,16#4C0,16#6C0;*)
	*)
END_VAR
IF Enable AND NOT Done THEN

	(*########################################################

		Configuration of CANopenSlave (Phoenix ILB CO DI16 DO16)
		
	#########################################################

		TransmissionType for TxPDOs and RxPDOs:

			0:										Event controlled and sychron (with SYNC-Object)
			1-240:									Cyclic and synchron (with SYNC-Object)
			254:									Producer specified
			255:									Acyclic and eventcontrolled 
			255 and EventTime = InhibitTime:	Cyclic

	#########################################################	*)


	(*************************************************** TxPDOs of CANOpenSlave ( MOVI-PLC ReceiveObjects) ***********************************************************)

	ExtConfig.NumberOfTxPDO				:= 1;		(*  TxPDO ---> CANopenSlave Transmit *)

	ExtConfig.TxPDO[1].EventTime			:= 0;		(* Slave: Index 0x18xx SubIndex 5: CycleTime in ms for CANopenSlave TXPDO *)
	ExtConfig.TxPDO[1].InhibitTime			:= 0;		(* Slave: Index 0x18xx SubIndex 3: InhibitTime in ms for CANopenSlave TxPDO *)
	ExtConfig.TxPDO[1].TransmissionType	:= 255;		(* Slave: Index 0x18xx SubIndex 2: TransmissionType for this TxPDO *)


	(*************************************************** RxPDOs of CANOpenSlave ( MOVI-PLC TransmitObjects) **********************************************************)

	ExtConfig.NumberOfRxPDO				:= 1;		(*  RxPDO ---> CANopenSlave Receive *)

	ExtConfig.RxPDO[1].EventTime			:= 0;		(* Master: CycleTime in ms for TransmitObjects (MOVI-PLC) *)
	ExtConfig.RxPDO[1].InhibitTime			:= 0;		(* Master: InhibitTime in ms for TransmitObjects (MOVI-PLC) *)
	ExtConfig.RxPDO[1].Length				:= 2;		(* Master: Length of this TransmitObject in bytes *)
	ExtConfig.RxPDO[1].TransmissionType	:= 255;		(* Slave: Index 0x14xx SubIndex 2: TransmissionType for this RxPDO *)


	(***************************************************** Additional parameters to set in the CANOpenSlave  ***************************************************************)

(*	Example to write user defined parameters (i.e. Index 16#6200):
	
	ExtConfig.stInitialParameter_COSlave.aIndex[1]			:= 16#6200;
	ExtConfig.stInitialParameter_COSlave.aSubIndex[1]	:= 0;
	ExtConfig.stInitialParameter_COSlave.aBytes[1]		:= 1;
	ExtConfig.stInitialParameter_COSlave.aData[1]			:= 16#64;
*)

	(********************************************** Additional configuration. Default values are in most cases sufficient *****************************************************)

	ExtConfig.bIOHold						:= FALSE;
	ExtConfig.bNoSettingsDownload			:= FALSE;
	ExtConfig.bWaitBeforeOperational		:= FALSE;
	ExtConfig.bResetUnconditional			:= FALSE;

	ExtConfig.TimeOutHeartBeat				:= 0;				(* [ms] *)
	ExtConfig.TimeOutNodeGuarding		:= 400;				(* [ms]. CAUTION ! DHP11B (MOVI-PLC basic) does NOT support NodeGuarding *)
	ExtConfig.TimeOutInitSequence			:= 6;				(* [seconds]. If the Init-Sequence takes longer than this TimeOut time --> Error *)
	ExtConfig.SyncCOBID						:= 0;				(* SyncObject ID for TransmissionType 0-240 (RxPDO). Usually 128. If 0, the ID will not be written *)
	ExtConfig.SyncTime						:= 0;				(* CycleTime for the SYNC-Object *)

	ExtConfig.TxPDO[1].COBID				:= 16#180;			(* In order to disable the use of RTR frames for the PDOs, set bit 30 = "RTR not allowed" *)
	ExtConfig.TxPDO[2].COBID				:= 16#280;			(* Ex. 16#4000_0280 *)
	ExtConfig.TxPDO[3].COBID				:= 16#380;
	ExtConfig.TxPDO[4].COBID				:= 16#480;			(* NOTE! These values are base values. The input "Address" will automatically be added *)
	ExtConfig.TxPDO[5].COBID				:= 16#680;
	ExtConfig.TxPDO[6].COBID				:= 16#1C0;
	ExtConfig.TxPDO[7].COBID				:= 16#2C0;
	ExtConfig.TxPDO[8].COBID				:= 16#3C0;
	ExtConfig.TxPDO[9].COBID				:= 16#4C0;
	ExtConfig.TxPDO[10].COBID				:= 16#6C0;

	ExtConfig.RxPDO[1].COBID				:= 16#200;
	ExtConfig.RxPDO[2].COBID				:= 16#300;
	ExtConfig.RxPDO[3].COBID				:= 16#400;
	ExtConfig.RxPDO[4].COBID				:= 16#500;
	ExtConfig.RxPDO[5].COBID				:= 16#780;
	ExtConfig.RxPDO[6].COBID				:= 16#240;
	ExtConfig.RxPDO[7].COBID				:= 16#340;
	ExtConfig.RxPDO[8].COBID				:= 16#440;
	ExtConfig.RxPDO[9].COBID				:= 16#540;
	ExtConfig.RxPDO[10].COBID				:= 16#7C0;

	Done := TRUE;

END_IF
END_FUNCTION_BLOCK

(* POU CodeSamples/CANopen/UniversalMaster/FB_Configuration_CANopenSlave_PNOZ, ST *)
FUNCTION_BLOCK FB_Configuration_CANopenSlave_PNOZ
VAR_INPUT
	Enable: BOOL; 			(* Activate config *)
END_VAR
VAR_OUTPUT
	Done: BOOL;				(* Config done *)
END_VAR
VAR_IN_OUT
	ExtConfig : MC_EXTENDEDCONFIG_COSLAVE	;
	(*
		########################################################################################################
			MC_EXTENDEDCONFIG_COSLAVE
		#########################################################################################################

						
		Variable								Value			Description
		-------------------------------------------------------------------------------------------------------------------------------------------------------------
		bWaitBeforeOperational 				BOOL;			When TRUE, after the coupler has been parameterized, it won't be switched in operational
																before this variable is FALSE. This can be used for example, to store the configuration with the FB
																MPLC_Universal_CANopen, with Service "SEWIOS_STORE", after a reset of the coppler 
		-------------------------------------------------------------------------------------------------------------------------------------------------------------
		bNoSettingsDownload 				BOOL;			TRUE : No configuration of the module. The configuration has to be done manually.
		-------------------------------------------------------------------------------------------------------------------------------------------------------------
		bResetUnconditional 					BOOL;			Even if the Connect FB isn't in fault it is possible to reset the bus coppler
		-------------------------------------------------------------------------------------------------------------------------------------------------------------
		bIOHold 								BOOL;			TRUE : Input data remain unchanged and the output data are not resetet also if the FB is in fault 
		-------------------------------------------------------------------------------------------------------------------------------------------------------------
		TimeOutHeartBeat					UINT;			If this value (ms) is different to zero, HeartbeatMode will be activated
		-------------------------------------------------------------------------------------------------------------------------------------------------------------
		TimeOutNodeGuarding 				UINT;			If this value (ms) is different to zero, NodeGuarding will be activated. 
																Caution ! The MOVI-PLC basic doesn´t support NodeGuarding 
		-------------------------------------------------------------------------------------------------------------------------------------------------------------
		TimeOutInitSequence					UINT;			Timeout for initialisation sequence (seconds) 
		-------------------------------------------------------------------------------------------------------------------------------------------------------------
		NumberOfRxPDO 					UINT;			Receive PDO : MOVI-PLC --> Slave  max. 32 
		-------------------------------------------------------------------------------------------------------------------------------------------------------------
		NumberOfTxPDO 						UINT;			Send PDO :      Slave --> MOVI-PLC  max 32 
		-------------------------------------------------------------------------------------------------------------------------------------------------------------	
		SyncTime 								USINT;			Cycle time of the sync telegram in ms. 
																Default = 0 : no sync will be started.
																If  SyncTime > 0, this FB initializes a sync telegram with the ID set at SyncCOBID. 
																The slave has to support synchronous communication 
		-------------------------------------------------------------------------------------------------------------------------------------------------------------
		SyncCOBID							UINT;			Index 1005h. ID of the sync telegram. Usually 16#80. IF 0, the ID won't be written.
		-------------------------------------------------------------------------------------------------------------------------------------------------------------
		SyncTimeOut 							INT := -1;		Index 1006h. Normally equal to SyncTime. 
																The slave usually set SyncTimeOut equal to SyncTime * 1.5. 
																If < 0, the index won't be written. 0 means no control over the sync interval 
		-------------------------------------------------------------------------------------------------------------------------------------------------------------
		stInitialParameter_COSlave 			MC_INITIALPARAMETER_COSLAVE;
												(*#################################################################
												With this struct, user defined parameters will be written to the BusCoupler after the
												initialization of the MPLC_ConnectUniversalSlave_CANopen. 
												Add the following code to your program to initialise the struct : 
												Example:
												Index 16#6423:	Activates the event-driven transmission of PDOs with analog inputs
												Index 16#3500:	Index from the manufacturer specific profile area
	
													stInitialParameter_COSlave.aIndex[1] := 16#6423;  	(* Index to write to *)
													stInitialParameter_COSlave.aSubIndex[1] := 0;   	(* SubIndex to write to *)
													stInitialParameter_COSlave.aBytes[1] := 1;   		(* Number of bytes to write  *)
													stInitialParameter_COSlave.aData[1] := 1;   			(* Data *)
	
													stInitialParameter_COSlave.aIndex[2] := 16#3500;  	(* Index to write to *)
													stInitialParameter_COSlave.aSubIndex[2] := 0;   	(* SubIndex to write to *)
													stInitialParameter_COSlave.aBytes[2] := 2;   		(* Number of bytes to write *)
													stInitialParameter_COSlave.aData[2] := 5;   			(* Data *)
	
												If there are more than 10 (DHP11B) or 64 (DHx41B) parameters to write, declare 
												NUMOF_INITIALPARAMETER in your program.
	
													VAR_GLOBAL CONSTANT
														NUMOF_INITIALPARAMETER : UDINT := 20;	
													END_VAR
	
												##################################################################*)
			-------------------------------------------------------------------------------------------------------------------------------------------------------------
		(* IDs of the PDO telegrams. The IDs are always calculated with the following IDs as a basis + the address of the bus coupler *)

		RxPDO 								ARRAY[1..32] OF MC_PDO_COSLAVE;			(* MOVI-PLC --> Slave *)
												(* := 16#200,16#300,16#400,16#500,16#780,16#240,16#340,16#440,16#540,16#7C0;	*)
		-------------------------------------------------------------------------------------------------------------------------------------------------------------
		TxPDO 								ARRAY[1..32] OF MC_PDO_COSLAVE; 			(* Slave --> MOVI-PLC *)
												(*:= 16#180,16#280,16#380,16#480,16#680,16#1C0,16#2C0,16#3C0,16#4C0,16#6C0;*)
	*)
END_VAR
(* 21.12.2010	FL  noch nicht getestet *)


IF Enable AND NOT Done THEN

	(*########################################################

		Configuration of CANopenSlave PNOZ)
		
		NOTE! 
		
	#########################################################

		TransmissionType for TxPDOs and RxPDOs:

			0:										Event controlled and sychron (with SYNC-Object)
			1-240:									Cyclic and synchron (with SYNC-Object)
			254:									Producer specified
			255:									Acyclic and eventcontrolled 
			255 and EventTime = InhibitTime:	Cyclic

	#########################################################	*)

	ExtConfig.bWaitBeforeOperational			:=FALSE;
	ExtConfig.bNoSettingsDownload				:=FALSE;
	ExtConfig.bResetUnconditional				:=FALSE;
	ExtConfig.bIOHold 							:=FALSE;

	ExtConfig.TimeOutHeartBeat 				:=16#FFFF;
	ExtConfig.TimeOutNodeGuarding 			:=16#00;
	ExtConfig.TimeOutInitSequence 				:=16#10;

	ExtConfig.SyncCOBID							:= 128;				(* SyncObject ID for TransmissionType 0-240 (RxPDO). Usually 128. If 0, the ID will not be written *)
	ExtConfig.SyncTime							:= 0;				(* CycleTime for the SYNC-Object *)
	ExtConfig.SyncTimeOut 						:=-1;



	(**************************************************** TxPDOs of CANOpenSlave ( MOVI-PLC ReceiveObjects) ************************************************************)

	ExtConfig.NumberOfTxPDO		:= 3;		(*  TxPDO ---> CANopenSlave Transmit *)
(* TxPDO ---> Sende-PDO1:AusgangsDaten 0---7 *)
	ExtConfig.TxPDO[1].EventTime	:= 0;		(* Master: CycleTime in ms for TransmitObjects (MOVI-PLC) *)
	ExtConfig.TxPDO[1].Length		:= 8;		(* Master: Length of this TransmitObject in bytes *)
(*  TxPDO ---> Sende-PDO2: :AusgangsDaten 8---15 *)
	ExtConfig.TxPDO[2].EventTime	:= 0;		(* Master: CycleTime in ms for TransmitObjects (MOVI-PLC) *)
	ExtConfig.TxPDO[2].Length		:= 8;		(* Master: Length of this TransmitObject in bytes *)
(*  Sende PDO3: :AusgangsDaten 16---19  *)
	ExtConfig.TxPDO[3].EventTime	:= 0;		(* Master: CycleTime in ms for TransmitObjects (MOVI-PLC) *)
	ExtConfig.TxPDO[3].Length		:= 8;		(* Master: Length of this TransmitObject in bytes *)


	(*************************************************** RxPDOs of CANOpenSlave ( MOVI-PLC TransmitObjects) **********************************************************)
	ExtConfig.NumberOfRxPDO			:= 3;		(*  RxPDO ---> CANopenSlave Receive *)

	(* Empfangs-PDO: EingangsDaten 0---7 *)
	ExtConfig.RxPDO[1].InhibitTime		:= 0;		(* Master: InhibitTime in ms for TransmitObjects (MOVI-PLC) *)
	ExtConfig.RxPDO[1].Length			:= 8;		(* Master: Length of this TransmitObject in bytes *)

	(* Empfangs-PDO:EingangsDaten 8--15*)
	ExtConfig.RxPDO[2].InhibitTime		:= 0;		(* Master: InhibitTime in ms for TransmitObjects (MOVI-PLC) *)
	ExtConfig.RxPDO[2].Length			:= 8;		(* Master: Length of this TransmitObject in bytes *)
	(* Empfangs-PDO: EingangsDaten 16---19*)
	ExtConfig.RxPDO[3].InhibitTime		:= 0;		(* Master: InhibitTime in ms for TransmitObjects (MOVI-PLC) *)
	ExtConfig.RxPDO[3].Length			:= 8;		(* Master: Length of this TransmitObject in bytes *)


	(***************************************************** Additional parameters to set in the CANOpenSlave  ***************************************************************)

	(* Set rotation direction *)

	(********************************************** Additional configuration. Default values are in most cases sufficient *****************************************************)



	ExtConfig.TxPDO[1].COBID				:= 16#180;		(* Impossible to change*)
	ExtConfig.TxPDO[2].COBID				:= 16#280;		(* Impossible to change*)
	ExtConfig.TxPDO[3].COBID				:= 16#1C0;	(* Impossible to change*)

	ExtConfig.RxPDO[1].COBID				:= 16#200;		(* Impossible to change*)
	ExtConfig.RxPDO[2].COBID				:= 16#300;		(* Impossible to change*)
	ExtConfig.RxPDO[3].COBID				:= 16#240;		(* Impossible to change*)

	Done := TRUE;

END_IF
END_FUNCTION_BLOCK

(* POU CodeSamples/CANopen/UniversalMaster/FB_Configuration_CANopenSlave_SchneiderFTB, ST *)
FUNCTION_BLOCK FB_Configuration_CANopenSlave_SchneiderFTB
VAR_INPUT
	Enable: BOOL; 			(* Activate config *)
END_VAR
VAR_OUTPUT
	Done: BOOL;				(* Config done *)
END_VAR
VAR_IN_OUT
	ExtConfig : MC_EXTENDEDCONFIG_COSLAVE	;
	(*
		########################################################################################################
			MC_EXTENDEDCONFIG_COSLAVE
		#########################################################################################################

						
		Variable								Value			Description
		-------------------------------------------------------------------------------------------------------------------------------------------------------------
		bWaitBeforeOperational :				 BOOL;	(* when TRUE, after the coupler has been parameterized, it won't be switched in operational
															before this variable is FALSE. This can be used for example, to store the configuration with the FB
															MPLC_Universal_CANopen, with Service "SEWIOS_STORE", after a reset of the coppler *)
		bNoSettingsDownload : 				BOOL;	(* when TRUE, all the parameters won't be downloaded to the coupler. This may be the case, once
															the coupler has been parameterized, and as long as the configuration and the coupler are not changed,
															it is not necessary to do it anymore *)
		bResetUnconditional :				BOOL;	(* even if the Connect FB isn't in fault it is possible to reset the bus coppler *)
		bIOHold :								BOOL;	(* when TRUE, the input data remain unchanged and the output data are not resetet also if the FB is in fault *)
		TimeOutHeartBeat :					UINT;	(* It is possible to use the NodeGuarding OR the HeartbeatMode (not both together). If you want to use one Mode
											  			  Consumer Heartbeat in ms*)
		bNoHeartBeat_Consumer:			BOOL := FALSE; (*Index 1016 SubIndex 0 not available*)
		DivTimeOutHeartBeat:				UINT:=4;(*	IF HeartbeatMode is activate AND ProducerHeartbeat is avaible,
															the Heartbeat Producertime is TimeOutHearBeat / this value.*)
		bNoHeartBeat_Producer: 			BOOL := FALSE;(* Index 1017 SubIndex 0 not available *)
		TimeOutNodeGuarding :				UINT;	(* the corresponding Timeout - Value has to be set > 0 (in ms). Caution ! The MOVI-PLC basic doesn´t support the Node Guarding *)
		bNoNodeGuarding: 					BOOL:=FALSE;(* the Index of NodeGuarding isn`t available *)
		TimeOutInitSequence:				UINT;	(* Time in seconds *)
		NumberOfRxPDO :					UINT;	(* MOVI-PLC --> Slave, max. 32 *)
		NumberOfTxPDO :					UINT;	(* Slave --> MOVI-PLC, max 32 *)
		OffsetOfRxPDO:						UINT;	(* Offset for the 1. RxPDO *)
		OffsetOfTxPDO:						UINT;	(* Offset for the 1. TxPDO *)
	
		SyncTime :							USINT;	(* cycle time of the sync telegram in ms. Default = 0 : no sync will be started.
															If > 0, this FB initializes a sync telegram with the following ID (if not 0). The slave has to support synchronous communication *)
		SyncCOBID :							UINT;	(* Index 1005h. ID of the sync telegram. Usually 16#80. If 0, the ID won't be written. *)
		SyncTimeOut :							INT := -1;	(* Index 1006h. Normally egal to SyncTime. The slave makes usually itself *1.5. If  <0, the index won't be written.
																0 means no control over the sync interval *)
	
		stInitialParameter_COSlave : 		MC_INITIALPARAMETER_COSLAVE;
												(*#################################################################
												 With this struct, ten user defined parameters will be written to the axis during the
												 initialization of MPLC_ConnectCANopenSlave. 
												 Add the following code to your program to initialise the struct : 
												Example:
												Index 16#6423:	Activates the event-driven transmission of PDOs with analog inputs
												Index 16#3000:	Index from the manufacturer specific profile area
	
													stInitialParameter_COSlave.aIndex[1] := 16#6423;  	(* Index to write to *)
													stInitialParameter_COSlave.aSubIndex[1] := 0;   	(* SubIndex to write to *)
													stInitialParameter_COSlave.aBytes[1] := 1;   		(* Number of bytes to write  *)
													stInitialParameter_COSlave.aData[1] := 1;   		(* Data *)
	
													stInitialParameter_COSlave.aIndex[2] := 16#3000;  	(* Index to write to *)
													stInitialParameter_COSlave.aSubIndex[2] := 0;   	(* SubIndex to write to *)
													stInitialParameter_COSlave.aBytes[2] := 2;   		(* Number of bytes to write *)
													stInitialParameter_COSlave.aData[2] := 5;   			(* Data *)
	
												If there are more than 10 parameters to write, declare NUMOF_INITIALPARAMETER
												in your program.
	
													VAR_GLOBAL CONSTANT
														NUMOF_INITIALPARAMETER : UDINT := 20;	
													END_VAR
	
												##################################################################*)

		bNoDeactivatePDO:					BOOL := FALSE; (* Change of Transmission Type, Inhibit- and Event- Time without deactivate RxPDO and TxPDO*)
		bNoTransmissionTyp_TxPDO: 		BOOL := FALSE; (* Transmission Type for TxPDO not changeable *)
		bNoTransmissionTyp_RxPDO: 		BOOL:= FALSE; (* Transmission Type for RxPDO not changeable *)
		bNoChangeCOBID_TxPDO      : 		BOOL := FALSE; (* COBID for TxPDO not changeable *)
		bNoChangeCOBID_RxPDO     : 		BOOL := FALSE; (* COBID for RxPDO not changeable *)
	
		(* IDs of the PDO telegrams. The IDs are always calculated with the following IDs as a basis + the address of the bus coppler *)
		RxPDO : ARRAY[1..32] OF MC_PDO_COSLAVE;(* := 16#200,16#300,16#400,16#500,16#780,16#240,16#340,16#440,16#540,16#7C0;		(* MOVI-PLC --> Bus coppler *)*)
		TxPDO : ARRAY[1..32] OF MC_PDO_COSLAVE; (*:= 16#180,16#280,16#380,16#480,16#680,16#1C0,16#2C0,16#3C0,16#4C0,16#6C0;	(* Bus coppler --> MOVI-PLC *)*)
	*)
END_VAR
IF Enable AND NOT Done THEN

	(*########################################################

		Configuration of CANopenSlave Schneider FTB 1CN .........
		
	#########################################################

		TransmissionType for TxPDOs and RxPDOs:

			0:										Event controlled and sychron (with SYNC-Object)
			1-240:									Cyclic and synchron (with SYNC-Object)
			254:									Producer specified
			255:									Acyclic and eventcontrolled 
			255 and EventTime = InhibitTime:	Cyclic

	#########################################################	*)


	(*************************************************** TxPDOs of CANOpenSlave ( MOVI-PLC ReceiveObjects) ***********************************************************)

	ExtConfig.NumberOfTxPDO				:= 1;		(*  TxPDO ---> CANopenSlave Transmit *)

	ExtConfig.TxPDO[1].EventTime			:= 100;		(* Slave: Index 0x18xx SubIndex 5: CycleTime in ms for CANopenSlave TXPDO *)
	ExtConfig.TxPDO[1].InhibitTime			:= 10;		(* Slave: Index 0x18xx SubIndex 3: InhibitTime in ms for CANopenSlave TxPDO *)
	ExtConfig.TxPDO[1].TransmissionType	:= 255;		(* Slave: Index 0x18xx SubIndex 2: TransmissionType for this TxPDO *)




	(*************************************************** RxPDOs of CANOpenSlave ( MOVI-PLC TransmitObjects) **********************************************************)

	ExtConfig.NumberOfRxPDO				:= 1;		(*  RxPDO ---> CANopenSlave Receive *)

	ExtConfig.RxPDO[1].EventTime			:= 100;		(* Master: CycleTime in ms for TransmitObjects (MOVI-PLC) *)
	ExtConfig.RxPDO[1].InhibitTime			:= 10;		(* Master: InhibitTime in ms for TransmitObjects (MOVI-PLC) *)
	ExtConfig.RxPDO[1].Length				:= 8;		(* Master: Length of this TransmitObject in bytes *)
	ExtConfig.RxPDO[1].TransmissionType	:= 255;		(* Slave: Index 0x14xx SubIndex 2: TransmissionType for this RxPDO *)




	(***************************************************** Additional parameters to set in the CANOpenSlave  ***************************************************************)
(* Parameter for FTB 1CN *)
	ExtConfig.stInitialParameter_COSlave.aIndex[1]			:= 16#2000;(**)
	ExtConfig.stInitialParameter_COSlave.aSubIndex[1]	:= 1;(* Input function channel 10..17*)
	ExtConfig.stInitialParameter_COSlave.aBytes[1]		:= 1;
	ExtConfig.stInitialParameter_COSlave.aData[1]			:= 2#00000000;(* 0=Input, 1=Diag Input *)

	ExtConfig.stInitialParameter_COSlave.aIndex[2]			:= 16#2001;(**)
	ExtConfig.stInitialParameter_COSlave.aSubIndex[2]	:= 1;(* Inpu/Output selection, channel 0..7,  *)
	ExtConfig.stInitialParameter_COSlave.aBytes[2]		:= 1;
	ExtConfig.stInitialParameter_COSlave.aData[2]			:= 2#00000000;(* 0=Input, 1=Output *)

	ExtConfig.stInitialParameter_COSlave.aIndex[3]			:= 16#2001;(**)
	ExtConfig.stInitialParameter_COSlave.aSubIndex[3]	:= 2;(* Inpu/Output selection, channel 10..17,  *)
	ExtConfig.stInitialParameter_COSlave.aBytes[3]		:= 1;
	ExtConfig.stInitialParameter_COSlave.aData[3]			:= 2#00000000;(* 0=Input, 1=Output *)


	(********************************************** Additional configuration. Default values are in most cases sufficient *****************************************************)

	ExtConfig.bIOHold						:= FALSE;
	ExtConfig.bNoSettingsDownload			:= FALSE;
	ExtConfig.bWaitBeforeOperational		:= FALSE;
	ExtConfig.bResetUnconditional			:= FALSE;

	ExtConfig.TimeOutHeartBeat				:= 250;				(* [ms] *)
(*	ExtConfig.DivTimeOutHeartBeat			:= 2;				(* Heartbeat Consumer = ExtConfig.TimeOutHeartBeat	 / ExtConfig.DivTimeOutHeartBeat *)*)
	ExtConfig.TimeOutNodeGuarding		:= 0;				(* [ms]. CAUTION ! DHP11B (MOVI-PLC basic) does NOT support NodeGuarding *)
	ExtConfig.TimeOutInitSequence			:= 10;				(* [seconds]. If the Init-Sequence takes longer than this TimeOut time --> Error *)
	ExtConfig.SyncCOBID						:= 0;				(* SyncObject ID for TransmissionType 0-240 (RxPDO). Usually 128. If 0, the ID will not be written *)
	ExtConfig.SyncTime						:= 0;				(* CycleTime for the SYNC-Object *)

	ExtConfig.TxPDO[1].COBID				:= 16#180;			(* In order to disable the use of RTR frames for the PDOs, set bit 30 = "RTR not allowed" *)
	ExtConfig.TxPDO[2].COBID				:= 16#280;			(* Ex. 16#4000_0280 *)
	ExtConfig.TxPDO[3].COBID				:= 16#380;
	ExtConfig.TxPDO[4].COBID				:= 16#480;			(* NOTE! These values are base values. The input "Address" will automatically be added *)
	ExtConfig.TxPDO[5].COBID				:= 16#680;
	ExtConfig.TxPDO[6].COBID				:= 16#1C0;
	ExtConfig.TxPDO[7].COBID				:= 16#2C0;
	ExtConfig.TxPDO[8].COBID				:= 16#3C0;
	ExtConfig.TxPDO[9].COBID				:= 16#4C0;
	ExtConfig.TxPDO[10].COBID				:= 16#6C0;

	ExtConfig.RxPDO[1].COBID				:= 16#200;
	ExtConfig.RxPDO[2].COBID				:= 16#300;
	ExtConfig.RxPDO[3].COBID				:= 16#400;
	ExtConfig.RxPDO[4].COBID				:= 16#500;
	ExtConfig.RxPDO[5].COBID				:= 16#780;
	ExtConfig.RxPDO[6].COBID				:= 16#240;
	ExtConfig.RxPDO[7].COBID				:= 16#340;
	ExtConfig.RxPDO[8].COBID				:= 16#440;
	ExtConfig.RxPDO[9].COBID				:= 16#540;
	ExtConfig.RxPDO[10].COBID				:= 16#7C0;

	Done := TRUE;

END_IF
END_FUNCTION_BLOCK

(* POU CodeSamples/CANopen/UniversalMaster/FB_Configuration_CANopenSlave_SEW_OCC11B, ST *)
FUNCTION_BLOCK FB_Configuration_CANopenSlave_SEW_OCC11B
VAR_INPUT
	Enable: BOOL; 			(* Activate config *)
END_VAR
VAR_OUTPUT
	Done: BOOL;				(* Config done *)
END_VAR
VAR_IN_OUT
	ExtConfig : MC_EXTENDEDCONFIG_COSLAVE	;
	(*
		########################################################################################################
			MC_EXTENDEDCONFIG_COSLAVE
		#########################################################################################################

						
		Variable								Value			Description
		-------------------------------------------------------------------------------------------------------------------------------------------------------------
		bWaitBeforeOperational 				BOOL;			When TRUE, after the coupler has been parameterized, it won't be switched in operational
																before this variable is FALSE. This can be used for example, to store the configuration with the FB
																MPLC_Universal_CANopen, with Service "SEWIOS_STORE", after a reset of the coppler 
		-------------------------------------------------------------------------------------------------------------------------------------------------------------
		bNoSettingsDownload 				BOOL;			TRUE : No configuration of the module. The configuration has to be done manually.
		-------------------------------------------------------------------------------------------------------------------------------------------------------------
		bResetUnconditional 					BOOL;			Even if the Connect FB isn't in fault it is possible to reset the bus coppler
		-------------------------------------------------------------------------------------------------------------------------------------------------------------
		bIOHold 								BOOL;			TRUE : Input data remain unchanged and the output data are not resetet also if the FB is in fault 
		-------------------------------------------------------------------------------------------------------------------------------------------------------------
		TimeOutHeartBeat					UINT;			If this value (ms) is different to zero, HeartbeatMode will be activated
		-------------------------------------------------------------------------------------------------------------------------------------------------------------
		TimeOutNodeGuarding 				UINT;			If this value (ms) is different to zero, NodeGuarding will be activated. 
																Caution ! The MOVI-PLC basic doesn´t support NodeGuarding 
		-------------------------------------------------------------------------------------------------------------------------------------------------------------
		TimeOutInitSequence					UINT;			Timeout for initialisation sequence (seconds) 
		-------------------------------------------------------------------------------------------------------------------------------------------------------------
		NumberOfRxPDO 					UINT;			Receive PDO : MOVI-PLC --> Slave  max. 32 
		-------------------------------------------------------------------------------------------------------------------------------------------------------------
		NumberOfTxPDO 						UINT;			Send PDO :      Slave --> MOVI-PLC  max 32 
		-------------------------------------------------------------------------------------------------------------------------------------------------------------	
		SyncTime 								USINT;			Cycle time of the sync telegram in ms. 
																Default = 0 : no sync will be started.
																If  SyncTime > 0, this FB initializes a sync telegram with the ID set at SyncCOBID. 
																The slave has to support synchronous communication 
		-------------------------------------------------------------------------------------------------------------------------------------------------------------
		SyncCOBID							UINT;			Index 1005h. ID of the sync telegram. Usually 16#80. IF 0, the ID won't be written.
		-------------------------------------------------------------------------------------------------------------------------------------------------------------
		SyncTimeOut 							INT := -1;		Index 1006h. Normally equal to SyncTime. 
																The slave usually set SyncTimeOut equal to SyncTime * 1.5. 
																If < 0, the index won't be written. 0 means no control over the sync interval 
		-------------------------------------------------------------------------------------------------------------------------------------------------------------
		stInitialParameter_COSlave 			MC_INITIALPARAMETER_COSLAVE;
												(*#################################################################
												With this struct, user defined parameters will be written to the BusCoupler after the
												initialization of the MPLC_ConnectUniversalSlave_CANopen. 
												Add the following code to your program to initialise the struct : 
												Example:
												Index 16#6423:	Activates the event-driven transmission of PDOs with analog inputs
												Index 16#3500:	Index from the manufacturer specific profile area
	
													stInitialParameter_COSlave.aIndex[1] := 16#6423;  	(* Index to write to *)
													stInitialParameter_COSlave.aSubIndex[1] := 0;   	(* SubIndex to write to *)
													stInitialParameter_COSlave.aBytes[1] := 1;   		(* Number of bytes to write  *)
													stInitialParameter_COSlave.aData[1] := 1;   			(* Data *)
	
													stInitialParameter_COSlave.aIndex[2] := 16#3500;  	(* Index to write to *)
													stInitialParameter_COSlave.aSubIndex[2] := 0;   	(* SubIndex to write to *)
													stInitialParameter_COSlave.aBytes[2] := 2;   		(* Number of bytes to write *)
													stInitialParameter_COSlave.aData[2] := 5;   			(* Data *)
	
